// Mitsubishi GX Developer project: パレット取り外し   PLC: Q02

PROGRAM MAIN
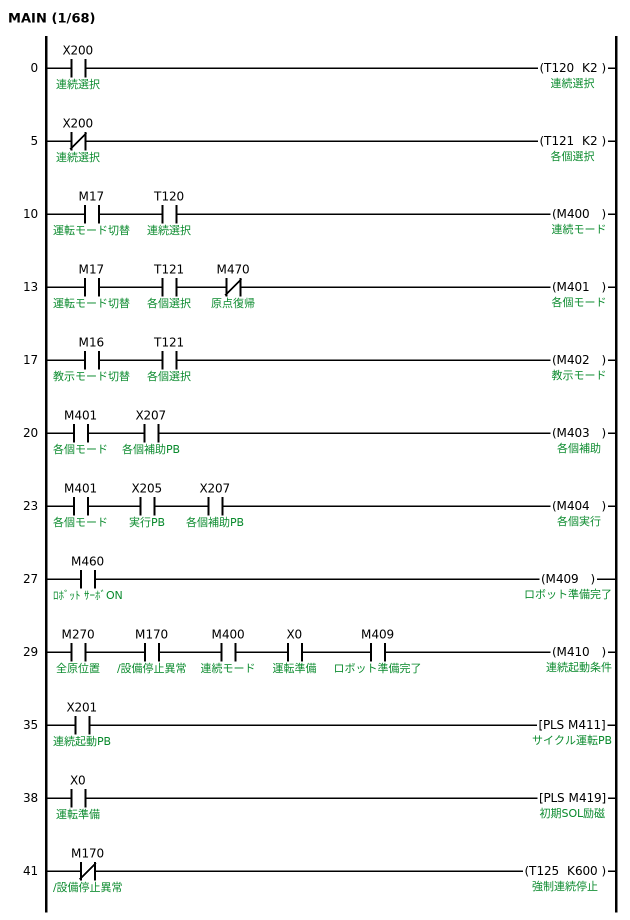
0     LD      X200  ; 連続選択
      OUT     T120 K2  ; 連続選択
5     LDI     X200  ; 連続選択
      OUT     T121 K2  ; 各個選択
10    LD      M17  ; 運転モード切替
      AND     T120  ; 連続選択
      OUT     M400  ; 連続モード
13    LD      M17  ; 運転モード切替
      AND     T121  ; 各個選択
      ANI     M470  ; 原点復帰
      OUT     M401  ; 各個モード
17    LD      M16  ; 教示モード切替
      AND     T121  ; 各個選択
      OUT     M402  ; 教示モード
20    LD      M401  ; 各個モード
      AND     X207  ; 各個補助PB
      OUT     M403  ; 各個補助
23    LD      M401  ; 各個モード
      AND     X205  ; 実行PB
      AND     X207  ; 各個補助PB
      OUT     M404  ; 各個実行
27    LD      M460  ; ﾛﾎﾞｯﾄ ｻｰﾎﾞON
      OUT     M409  ; ロボット準備完了
29    LD      M270  ; 全原位置
      AND     M170  ; /設備停止異常
      AND     M400  ; 連続モード
      AND     X0  ; 運転準備
      AND     M409  ; ロボット準備完了
      OUT     M410  ; 連続起動条件
35    LD      X201  ; 連続起動PB
      PLS     M411  ; サイクル運転PB
38    LD      X0  ; 運転準備
      PLS     M419  ; 初期SOL励磁
41    LDI     M170  ; /設備停止異常
      OUT     T125 K600  ; 強制連続停止
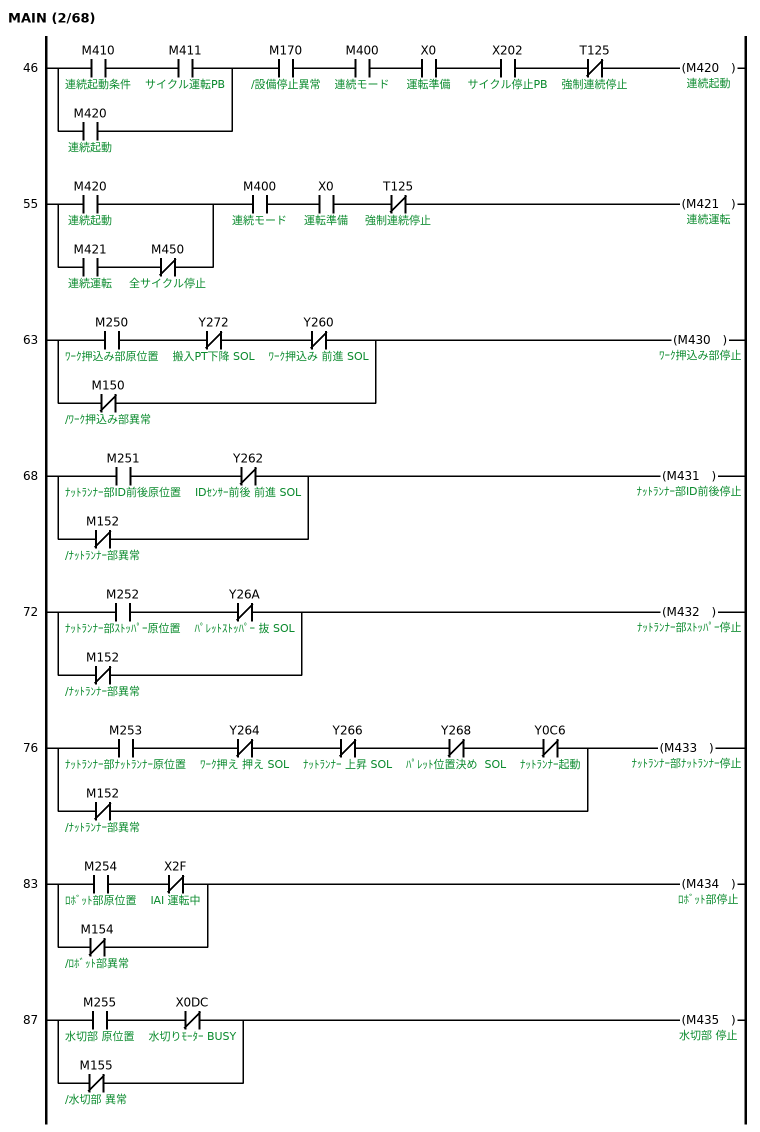
46    LD      M410  ; 連続起動条件
      AND     M411  ; サイクル運転PB
      OR      M420  ; 連続起動
      AND     M170  ; /設備停止異常
      AND     M400  ; 連続モード
      AND     X0  ; 運転準備
      AND     X202  ; サイクル停止PB
      ANI     T125  ; 強制連続停止
      OUT     M420  ; 連続起動
55    LD      M420  ; 連続起動
      LD      M421  ; 連続運転
      ANI     M450  ; 全サイクル停止
      ORB
      AND     M400  ; 連続モード
      AND     X0  ; 運転準備
      ANI     T125  ; 強制連続停止
      OUT     M421  ; 連続運転
63    LD      M250  ; ﾜｰｸ押込み部原位置
      ANI     Y272  ; 搬入PT下降 SOL
      ANI     Y260  ; ﾜｰｸ押込み 前進 SOL
      ORI     M150  ; /ﾜｰｸ押込み部異常
      OUT     M430  ; ﾜｰｸ押込み部停止
68    LD      M251  ; ﾅｯﾄﾗﾝﾅｰ部ID前後原位置
      ANI     Y262  ; IDｾﾝｻｰ前後 前進 SOL
      ORI     M152  ; /ﾅｯﾄﾗﾝﾅｰ部異常
      OUT     M431  ; ﾅｯﾄﾗﾝﾅｰ部ID前後停止
72    LD      M252  ; ﾅｯﾄﾗﾝﾅｰ部ｽﾄｯﾊﾟｰ原位置
      ANI     Y26A  ; ﾊﾟﾚｯﾄｽﾄｯﾊﾟｰ 抜 SOL
      ORI     M152  ; /ﾅｯﾄﾗﾝﾅｰ部異常
      OUT     M432  ; ﾅｯﾄﾗﾝﾅｰ部ｽﾄｯﾊﾟｰ停止
76    LD      M253  ; ﾅｯﾄﾗﾝﾅｰ部ﾅｯﾄﾗﾝﾅｰ原位置
      ANI     Y264  ; ﾜｰｸ押え 押え SOL
      ANI     Y266  ; ﾅｯﾄﾗﾝﾅｰ 上昇 SOL
      ANI     Y268  ; ﾊﾟﾚｯﾄ位置決め  SOL
      ANI     Y0C6  ; ﾅｯﾄﾗﾝﾅｰ起動
      ORI     M152  ; /ﾅｯﾄﾗﾝﾅｰ部異常
      OUT     M433  ; ﾅｯﾄﾗﾝﾅｰ部ﾅｯﾄﾗﾝﾅｰ停止
83    LD      M254  ; ﾛﾎﾞｯﾄ部原位置
      ANI     X2F  ; IAI 運転中
      ORI     M154  ; /ﾛﾎﾞｯﾄ部異常
      OUT     M434  ; ﾛﾎﾞｯﾄ部停止
87    LD      M255  ; 水切部 原位置
      ANI     X0DC  ; 水切りﾓｰﾀｰ BUSY
      ORI     M155  ; /水切部 異常
      OUT     M435  ; 水切部 停止
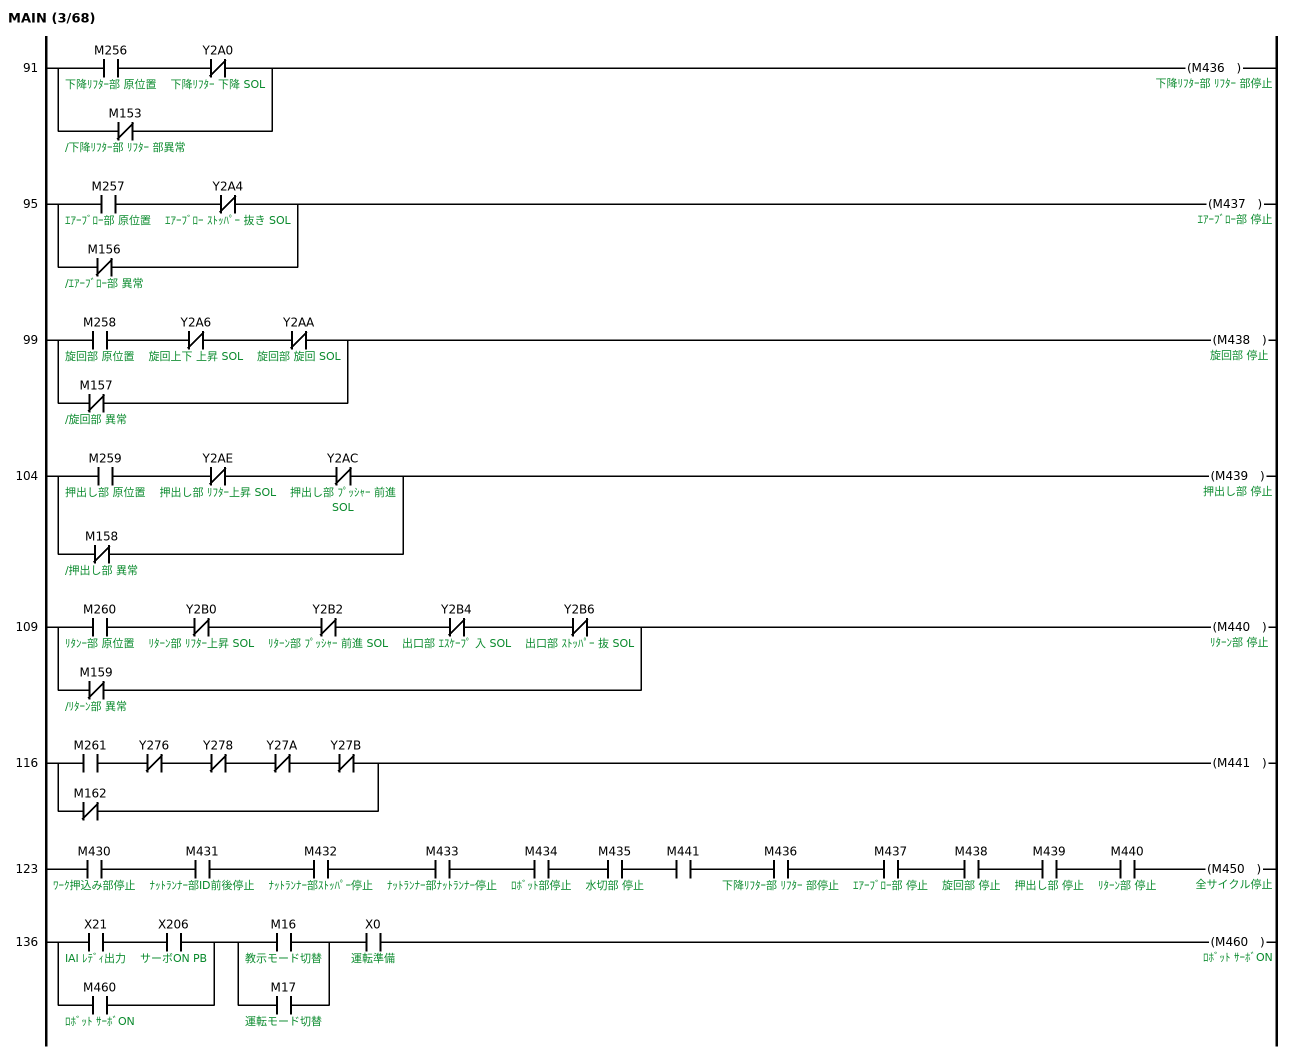
91    LD      M256  ; 下降ﾘﾌﾀｰ部 原位置
      ANI     Y2A0  ; 下降ﾘﾌﾀｰ 下降 SOL
      ORI     M153  ; /下降ﾘﾌﾀｰ部 ﾘﾌﾀｰ 部異常
      OUT     M436  ; 下降ﾘﾌﾀｰ部 ﾘﾌﾀｰ 部停止
95    LD      M257  ; ｴｱｰﾌﾞﾛｰ部 原位置
      ANI     Y2A4  ; ｴｱｰﾌﾞﾛｰ ｽﾄｯﾊﾟｰ 抜き SOL
      ORI     M156  ; /ｴｱｰﾌﾞﾛｰ部 異常
      OUT     M437  ; ｴｱｰﾌﾞﾛｰ部 停止
99    LD      M258  ; 旋回部 原位置
      ANI     Y2A6  ; 旋回上下 上昇 SOL
      ANI     Y2AA  ; 旋回部 旋回 SOL
      ORI     M157  ; /旋回部 異常
      OUT     M438  ; 旋回部 停止
104   LD      M259  ; 押出し部 原位置
      ANI     Y2AE  ; 押出し部 ﾘﾌﾀｰ上昇 SOL
      ANI     Y2AC  ; 押出し部 ﾌﾟｯｼｬｰ 前進 SOL
      ORI     M158  ; /押出し部 異常
      OUT     M439  ; 押出し部 停止
109   LD      M260  ; ﾘﾀﾝｰ部 原位置
      ANI     Y2B0  ; ﾘﾀｰﾝ部 ﾘﾌﾀｰ上昇 SOL
      ANI     Y2B2  ; ﾘﾀｰﾝ部 ﾌﾟｯｼｬｰ 前進 SOL
      ANI     Y2B4  ; 出口部 ｴｽｹｰﾌﾟ 入 SOL
      ANI     Y2B6  ; 出口部 ｽﾄｯﾊﾟｰ 抜 SOL
      ORI     M159  ; /ﾘﾀｰﾝ部 異常
      OUT     M440  ; ﾘﾀｰﾝ部 停止
116   LD      M261
      ANI     Y276
      ANI     Y278
      ANI     Y27A
      ANI     Y27B
      ORI     M162
      OUT     M441
123   LD      M430  ; ﾜｰｸ押込み部停止
      AND     M431  ; ﾅｯﾄﾗﾝﾅｰ部ID前後停止
      AND     M432  ; ﾅｯﾄﾗﾝﾅｰ部ｽﾄｯﾊﾟｰ停止
      AND     M433  ; ﾅｯﾄﾗﾝﾅｰ部ﾅｯﾄﾗﾝﾅｰ停止
      AND     M434  ; ﾛﾎﾞｯﾄ部停止
      AND     M435  ; 水切部 停止
      AND     M441
      AND     M436  ; 下降ﾘﾌﾀｰ部 ﾘﾌﾀｰ 部停止
      AND     M437  ; ｴｱｰﾌﾞﾛｰ部 停止
      AND     M438  ; 旋回部 停止
      AND     M439  ; 押出し部 停止
      AND     M440  ; ﾘﾀｰﾝ部 停止
      OUT     M450  ; 全サイクル停止
136   LD      X21  ; IAI ﾚﾃﾞｨ出力
      AND     X206  ; サーボON PB
      OR      M460  ; ﾛﾎﾞｯﾄ ｻｰﾎﾞON
      LD      M16  ; 教示モード切替
      OR      M17  ; 運転モード切替
      ANB
      AND     X0  ; 運転準備
      OUT     M460  ; ﾛﾎﾞｯﾄ ｻｰﾎﾞON
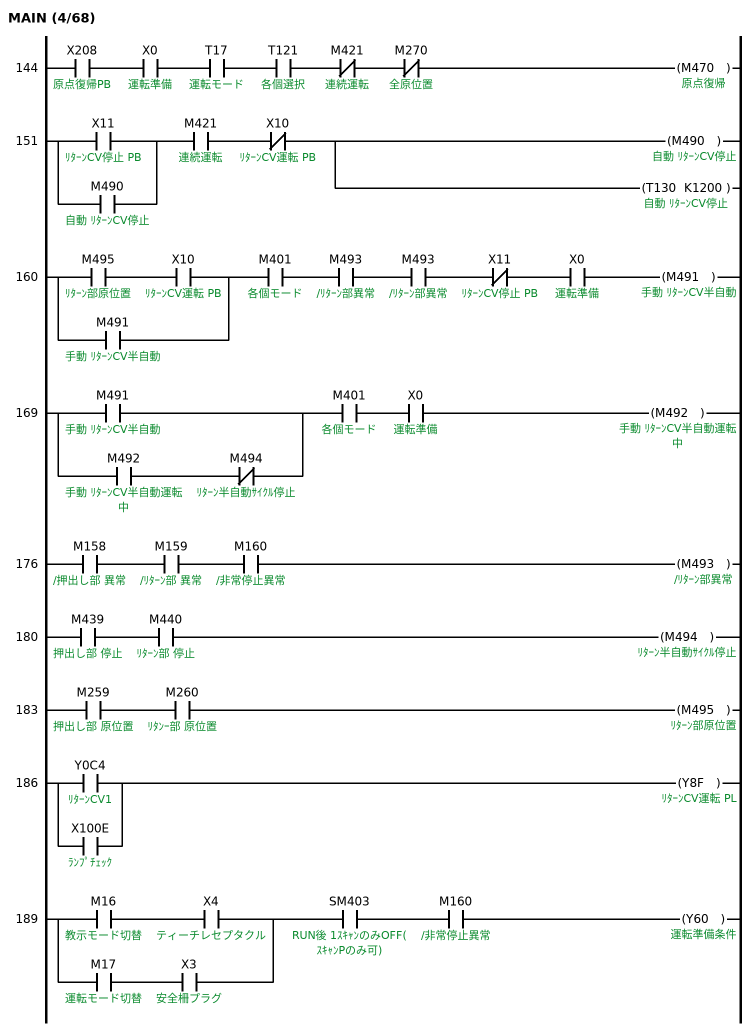
144   LD      X208  ; 原点復帰PB
      AND     X0  ; 運転準備
      AND     T17  ; 運転モード
      AND     T121  ; 各個選択
      ANI     M421  ; 連続運転
      ANI     M270  ; 全原位置
      OUT     M470  ; 原点復帰
151   LD      X11  ; ﾘﾀｰﾝCV停止 PB
      OR      M490  ; 自動 ﾘﾀｰﾝCV停止
      AND     M421  ; 連続運転
      ANI     X10  ; ﾘﾀｰﾝCV運転 PB
      OUT     M490  ; 自動 ﾘﾀｰﾝCV停止
      OUT     T130 K1200  ; 自動 ﾘﾀｰﾝCV停止
160   LD      M495  ; ﾘﾀｰﾝ部原位置
      AND     X10  ; ﾘﾀｰﾝCV運転 PB
      OR      M491  ; 手動 ﾘﾀｰﾝCV半自動
      AND     M401  ; 各個モード
      AND     M493  ; /ﾘﾀｰﾝ部異常
      AND     M493  ; /ﾘﾀｰﾝ部異常
      ANI     X11  ; ﾘﾀｰﾝCV停止 PB
      AND     X0  ; 運転準備
      OUT     M491  ; 手動 ﾘﾀｰﾝCV半自動
169   LD      M491  ; 手動 ﾘﾀｰﾝCV半自動
      LD      M492  ; 手動 ﾘﾀｰﾝCV半自動運転中
      ANI     M494  ; ﾘﾀｰﾝ半自動ｻｲｸﾙ停止
      ORB
      AND     M401  ; 各個モード
      AND     X0  ; 運転準備
      OUT     M492  ; 手動 ﾘﾀｰﾝCV半自動運転中
176   LD      M158  ; /押出し部 異常
      AND     M159  ; /ﾘﾀｰﾝ部 異常
      AND     M160  ; /非常停止異常
      OUT     M493  ; /ﾘﾀｰﾝ部異常
180   LD      M439  ; 押出し部 停止
      AND     M440  ; ﾘﾀｰﾝ部 停止
      OUT     M494  ; ﾘﾀｰﾝ半自動ｻｲｸﾙ停止
183   LD      M259  ; 押出し部 原位置
      AND     M260  ; ﾘﾀﾝｰ部 原位置
      OUT     M495  ; ﾘﾀｰﾝ部原位置
186   LD      Y0C4  ; ﾘﾀｰﾝCV1
      OR      X100E  ; ﾗﾝﾌﾟﾁｪｯｸ
      OUT     Y8F  ; ﾘﾀｰﾝCV運転 PL
189   LD      M16  ; 教示モード切替
      AND     X4  ; ティーチレセプタクル
      LD      M17  ; 運転モード切替
      AND     X3  ; 安全柵プラグ
      ORB
      AND     SM403  ; RUN後 1ｽｷｬﾝのみOFF(ｽｷｬﾝPのみ可)
      AND     M160  ; /非常停止異常
      OUT     Y60  ; 運転準備条件
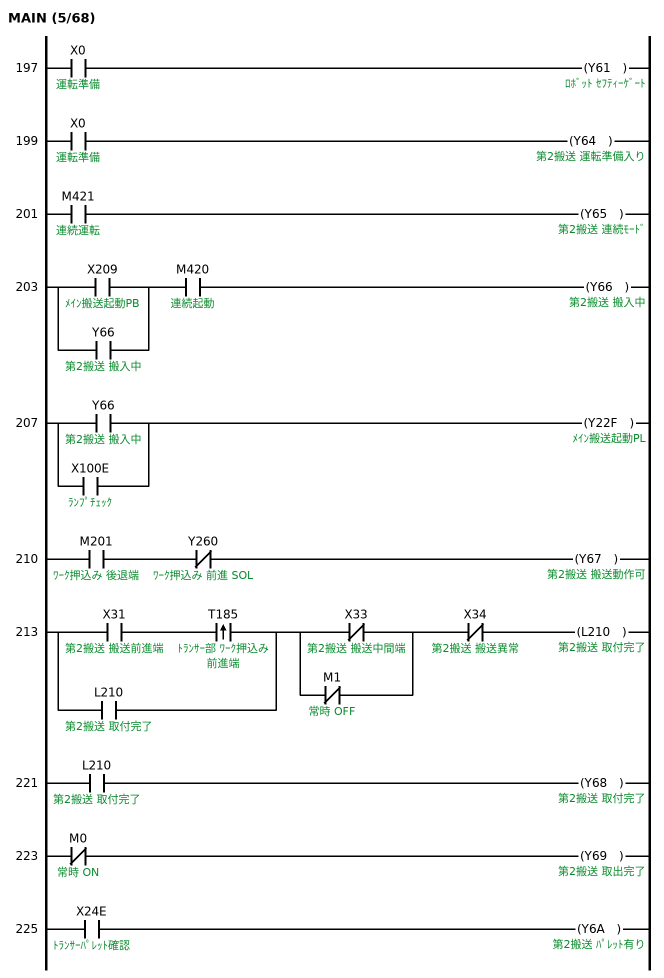
197   LD      X0  ; 運転準備
      OUT     Y61  ; ﾛﾎﾞｯﾄ ｾﾌﾃｨｰｹﾞｰﾄ
199   LD      X0  ; 運転準備
      OUT     Y64  ; 第2搬送 運転準備入り
201   LD      M421  ; 連続運転
      OUT     Y65  ; 第2搬送 連続ﾓｰﾄﾞ
203   LD      X209  ; ﾒｲﾝ搬送起動PB
      OR      Y66  ; 第2搬送 搬入中
      AND     M420  ; 連続起動
      OUT     Y66  ; 第2搬送 搬入中
207   LD      Y66  ; 第2搬送 搬入中
      OR      X100E  ; ﾗﾝﾌﾟﾁｪｯｸ
      OUT     Y22F  ; ﾒｲﾝ搬送起動PL
210   LD      M201  ; ﾜｰｸ押込み 後退端
      ANI     Y260  ; ﾜｰｸ押込み 前進 SOL
      OUT     Y67  ; 第2搬送 搬送動作可
213   LD      X31  ; 第2搬送 搬送前進端
      ANDP    T185  ; ﾄﾗﾝｻｰ部 ﾜｰｸ押込み 前進端
      OR      L210  ; 第2搬送 取付完了
      LDI     X33  ; 第2搬送 搬送中間端
      ORI     M1  ; 常時 OFF
      ANB
      ANI     X34  ; 第2搬送 搬送異常
      OUT     L210  ; 第2搬送 取付完了
221   LD      L210  ; 第2搬送 取付完了
      OUT     Y68  ; 第2搬送 取付完了
223   LDI     M0  ; 常時 ON
      OUT     Y69  ; 第2搬送 取出完了
225   LD      X24E  ; ﾄﾗﾝｻｰﾊﾟﾚｯﾄ確認
      OUT     Y6A  ; 第2搬送 ﾊﾟﾚｯﾄ有り
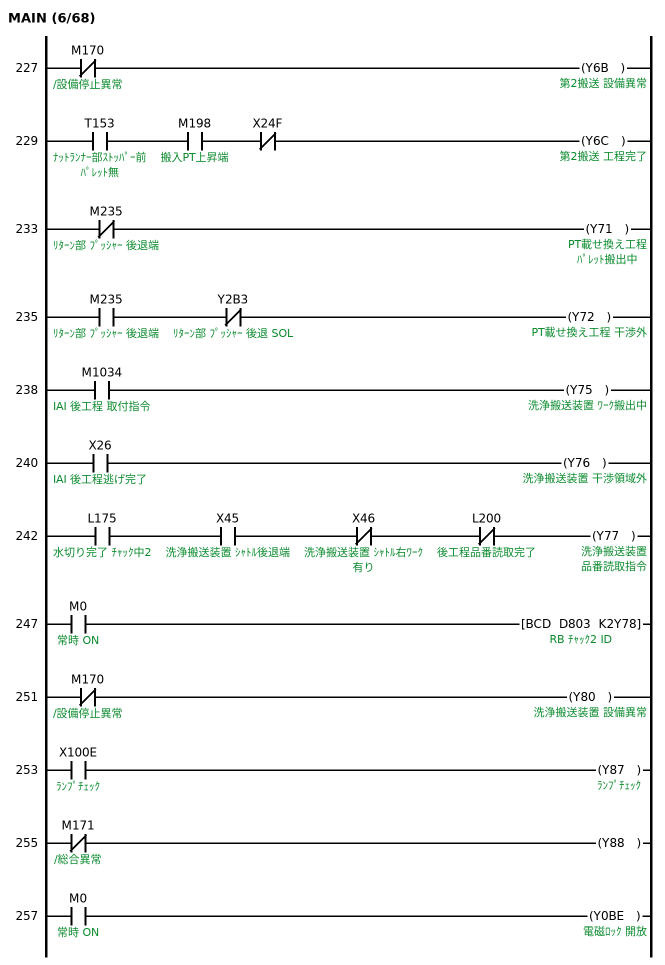
227   LDI     M170  ; /設備停止異常
      OUT     Y6B  ; 第2搬送 設備異常
229   LD      T153  ; ﾅｯﾄﾗﾝﾅｰ部ｽﾄｯﾊﾟｰ前 ﾊﾟﾚｯﾄ無
      AND     M198  ; 搬入PT上昇端
      ANI     X24F
      OUT     Y6C  ; 第2搬送 工程完了
233   LDI     M235  ; ﾘﾀｰﾝ部 ﾌﾟｯｼｬｰ 後退端
      OUT     Y71  ; PT載せ換え工程 ﾊﾟﾚｯﾄ搬出中
235   LD      M235  ; ﾘﾀｰﾝ部 ﾌﾟｯｼｬｰ 後退端
      ANI     Y2B3  ; ﾘﾀｰﾝ部 ﾌﾟｯｼｬｰ 後退 SOL
      OUT     Y72  ; PT載せ換え工程 干渉外
238   LD      M1034  ; IAI 後工程 取付指令
      OUT     Y75  ; 洗浄搬送装置 ﾜｰｸ搬出中
240   LD      X26  ; IAI 後工程逃げ完了
      OUT     Y76  ; 洗浄搬送装置 干渉領域外
242   LD      L175  ; 水切り完了 ﾁｬｯｸ中2
      AND     X45  ; 洗浄搬送装置 ｼｬﾄﾙ後退端
      ANI     X46  ; 洗浄搬送装置 ｼｬﾄﾙ右ﾜｰｸ有り
      ANI     L200  ; 後工程品番読取完了
      OUT     Y77  ; 洗浄搬送装置 品番読取指令
247   LD      M0  ; 常時 ON
      BCD     D803 K2Y78  ; RB ﾁｬｯｸ2 ID / 洗浄搬送装置 品番情報1
251   LDI     M170  ; /設備停止異常
      OUT     Y80  ; 洗浄搬送装置 設備異常
253   LD      X100E  ; ﾗﾝﾌﾟﾁｪｯｸ
      OUT     Y87  ; ﾗﾝﾌﾟﾁｪｯｸ
255   LDI     M171  ; /総合異常
      OUT     Y88
257   LD      M0  ; 常時 ON
      OUT     Y0BE  ; 電磁ﾛｯｸ 開放
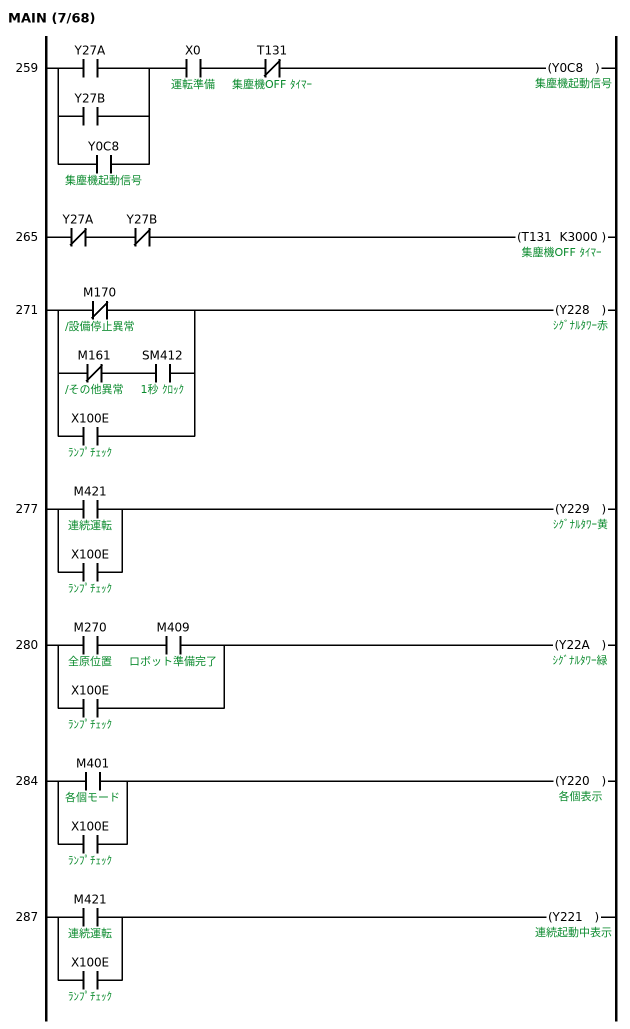
259   LD      Y27A
      OR      Y27B
      OR      Y0C8  ; 集塵機起動信号
      AND     X0  ; 運転準備
      ANI     T131  ; 集塵機OFF ﾀｲﾏｰ
      OUT     Y0C8  ; 集塵機起動信号
265   LDI     Y27A
      ANI     Y27B
      OUT     T131 K3000  ; 集塵機OFF ﾀｲﾏｰ
271   LDI     M170  ; /設備停止異常
      LDI     M161  ; /その他異常
      AND     SM412  ; 1秒 ｸﾛｯｸ
      ORB
      OR      X100E  ; ﾗﾝﾌﾟﾁｪｯｸ
      OUT     Y228  ; ｼｸﾞﾅﾙﾀﾜｰ赤
277   LD      M421  ; 連続運転
      OR      X100E  ; ﾗﾝﾌﾟﾁｪｯｸ
      OUT     Y229  ; ｼｸﾞﾅﾙﾀﾜｰ黄
280   LD      M270  ; 全原位置
      AND     M409  ; ロボット準備完了
      OR      X100E  ; ﾗﾝﾌﾟﾁｪｯｸ
      OUT     Y22A  ; ｼｸﾞﾅﾙﾀﾜｰ緑
284   LD      M401  ; 各個モード
      OR      X100E  ; ﾗﾝﾌﾟﾁｪｯｸ
      OUT     Y220  ; 各個表示
287   LD      M421  ; 連続運転
      OR      X100E  ; ﾗﾝﾌﾟﾁｪｯｸ
      OUT     Y221  ; 連続起動中表示
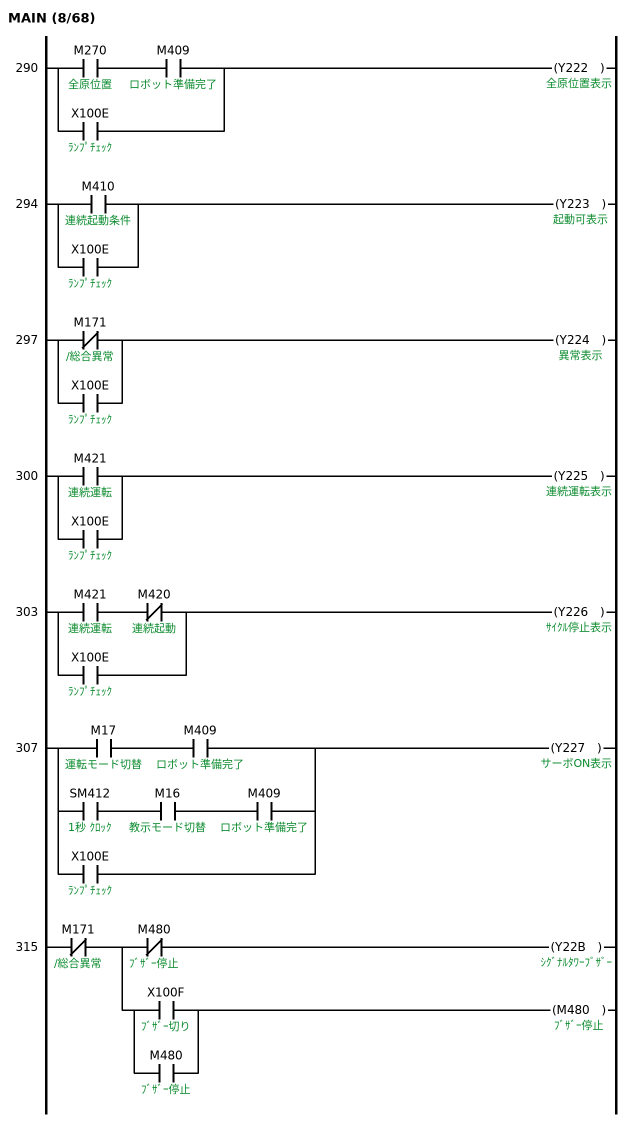
290   LD      M270  ; 全原位置
      AND     M409  ; ロボット準備完了
      OR      X100E  ; ﾗﾝﾌﾟﾁｪｯｸ
      OUT     Y222  ; 全原位置表示
294   LD      M410  ; 連続起動条件
      OR      X100E  ; ﾗﾝﾌﾟﾁｪｯｸ
      OUT     Y223  ; 起動可表示
297   LDI     M171  ; /総合異常
      OR      X100E  ; ﾗﾝﾌﾟﾁｪｯｸ
      OUT     Y224  ; 異常表示
300   LD      M421  ; 連続運転
      OR      X100E  ; ﾗﾝﾌﾟﾁｪｯｸ
      OUT     Y225  ; 連続運転表示
303   LD      M421  ; 連続運転
      ANI     M420  ; 連続起動
      OR      X100E  ; ﾗﾝﾌﾟﾁｪｯｸ
      OUT     Y226  ; ｻｲｸﾙ停止表示
307   LD      M17  ; 運転モード切替
      AND     M409  ; ロボット準備完了
      LD      SM412  ; 1秒 ｸﾛｯｸ
      AND     M16  ; 教示モード切替
      AND     M409  ; ロボット準備完了
      ORB
      OR      X100E  ; ﾗﾝﾌﾟﾁｪｯｸ
      OUT     Y227  ; サーボON表示
315   LDI     M171  ; /総合異常
      MPS
      ANI     M480  ; ﾌﾞｻﾞｰ停止
      OUT     Y22B  ; ｼｸﾞﾅﾙﾀﾜｰﾌﾞｻﾞｰ
      MPP
      LD      X100F  ; ﾌﾞｻﾞｰ切り
      OR      M480  ; ﾌﾞｻﾞｰ停止
      ANB
      OUT     M480  ; ﾌﾞｻﾞｰ停止
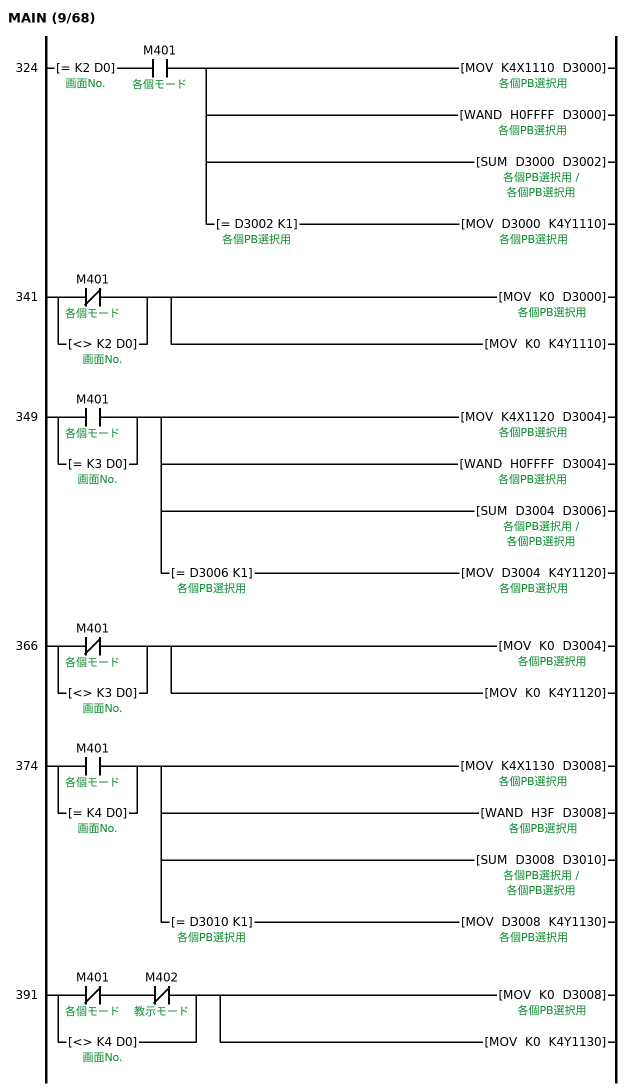
324   LD=     K2 D0  ; 画面No.
      AND     M401  ; 各個モード
      MOV     K4X1110 D3000  ; ﾜｰｸ押込み 後退 PB / 各個PB選択用
      WAND    H0FFFF D3000
      SUM     D3000 D3002  ; 各個PB選択用
      AND=    D3002 K1  ; 各個PB選択用
      MOV     D3000 K4Y1110  ; ﾜｰｸ押込み 後退 選択PL
341   LDI     M401  ; 各個モード
      OR<>    K2 D0  ; 画面No.
      MOV     K0 D3000
      MOV     K0 K4Y1110
349   LD      M401  ; 各個モード
      OR=     K3 D0  ; 画面No.
      MOV     K4X1120 D3004  ; 下降ﾘﾌﾀｰ部 ﾘﾌﾀｰ下降 PB / 各個PB選択用
      WAND    H0FFFF D3004
      SUM     D3004 D3006  ; 各個PB選択用
      AND=    D3006 K1  ; 各個PB選択用
      MOV     D3004 K4Y1120  ; 下降ﾘﾌﾀｰ部 ﾘﾌﾀｰ下降 選択PL
366   LDI     M401  ; 各個モード
      OR<>    K3 D0  ; 画面No.
      MOV     K0 D3004
      MOV     K0 K4Y1120
374   LD      M401  ; 各個モード
      OR=     K4 D0  ; 画面No.
      MOV     K4X1130 D3008  ; ﾛﾎﾞｯﾄ部 ﾁｬｯｸ1開 PB / 各個PB選択用
      WAND    H3F D3008
      SUM     D3008 D3010  ; 各個PB選択用
      AND=    D3010 K1  ; 各個PB選択用
      MOV     D3008 K4Y1130  ; ﾛﾎﾞｯﾄ部 ﾁｬｯｸ1開 選択PL
391   LDI     M401  ; 各個モード
      ANI     M402  ; 教示モード
      OR<>    K4 D0  ; 画面No.
      MOV     K0 D3008
      MOV     K0 K4Y1130
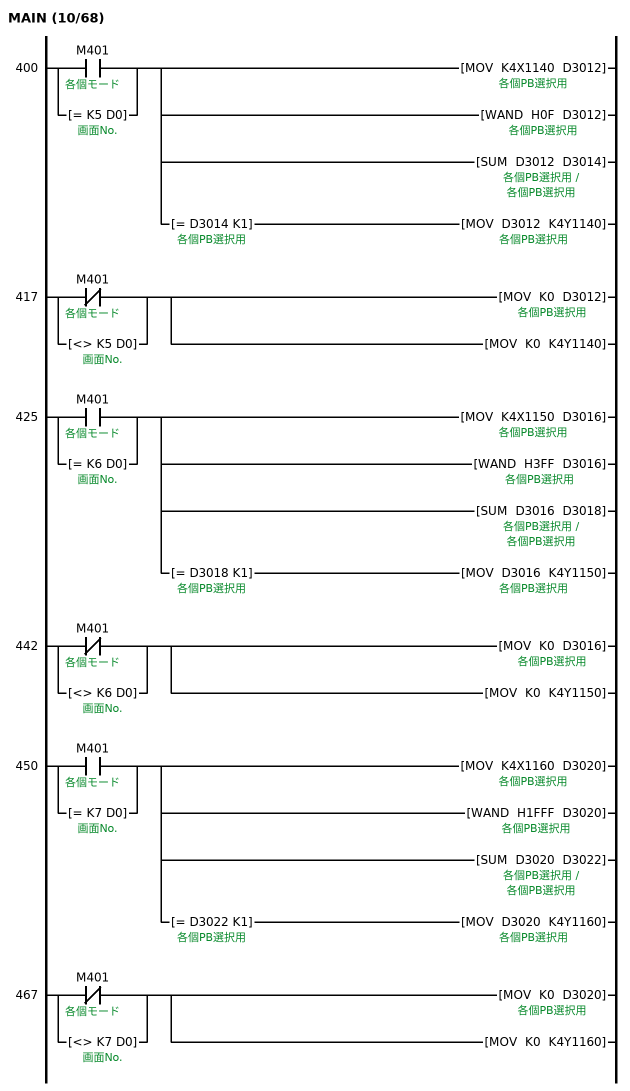
400   LD      M401  ; 各個モード
      OR=     K5 D0  ; 画面No.
      MOV     K4X1140 D3012  ; 水切部 ｼｬｯﾀｰ開 PB / 各個PB選択用
      WAND    H0F D3012
      SUM     D3012 D3014  ; 各個PB選択用
      AND=    D3014 K1  ; 各個PB選択用
      MOV     D3012 K4Y1140  ; 水切部 ｼｬｯﾀｰ開 選択PL
417   LDI     M401  ; 各個モード
      OR<>    K5 D0  ; 画面No.
      MOV     K0 D3012
      MOV     K0 K4Y1140
425   LD      M401  ; 各個モード
      OR=     K6 D0  ; 画面No.
      MOV     K4X1150 D3016  ; ｴｱｰﾌﾞﾛｰ ｼｬｯﾀｰ 開 PB / 各個PB選択用
      WAND    H3FF D3016
      SUM     D3016 D3018  ; 各個PB選択用
      AND=    D3018 K1  ; 各個PB選択用
      MOV     D3016 K4Y1150  ; ｴｱｰﾌﾞﾛｰ ｼｬｯﾀｰ 開 選択PL
442   LDI     M401  ; 各個モード
      OR<>    K6 D0  ; 画面No.
      MOV     K0 D3016
      MOV     K0 K4Y1150
450   LD      M401  ; 各個モード
      OR=     K7 D0  ; 画面No.
      MOV     K4X1160 D3020  ; 押出し部 ﾘﾌﾀｰ下降PB / 各個PB選択用
      WAND    H1FFF D3020
      SUM     D3020 D3022  ; 各個PB選択用
      AND=    D3022 K1  ; 各個PB選択用
      MOV     D3020 K4Y1160  ; 押出し部 ﾘﾌﾀｰ下降選択PL
467   LDI     M401  ; 各個モード
      OR<>    K7 D0  ; 画面No.
      MOV     K0 D3020
      MOV     K0 K4Y1160
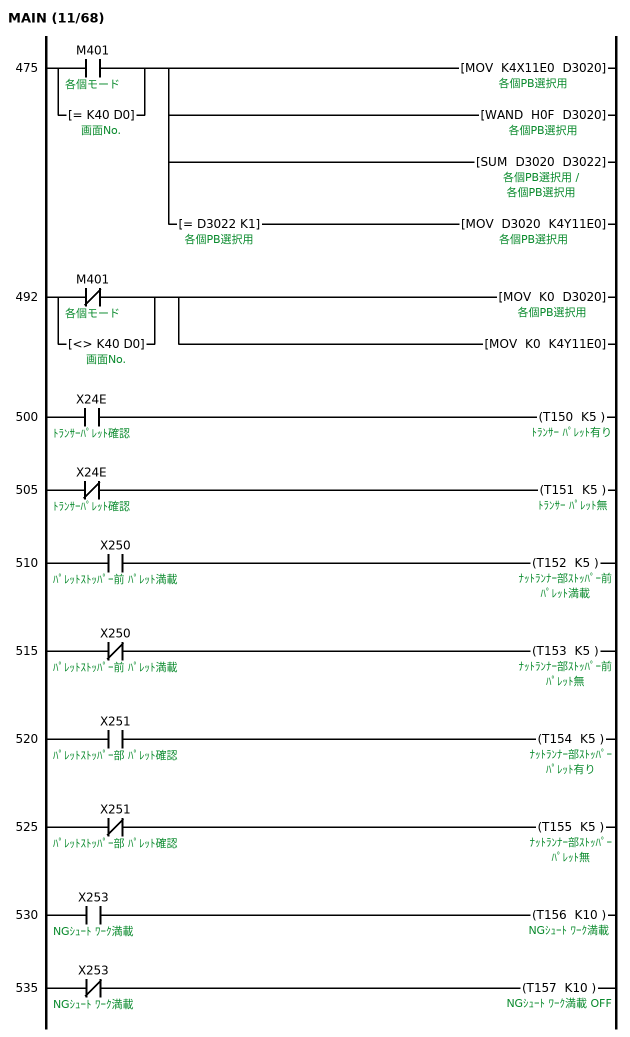
475   LD      M401  ; 各個モード
      OR=     K40 D0  ; 画面No.
      MOV     K4X11E0 D3020  ; ID読出し PB
      WAND    H0F D3020
      SUM     D3020 D3022
      AND=    D3022 K1  ; 各個PB選択用
      MOV     D3020 K4Y11E0  ; ID読出し 選択PL
492   LDI     M401  ; 各個モード
      OR<>    K40 D0  ; 画面No.
      MOV     K0 D3020
      MOV     K0 K4Y11E0
500   LD      X24E  ; ﾄﾗﾝｻｰﾊﾟﾚｯﾄ確認
      OUT     T150 K5  ; ﾄﾗﾝｻｰ ﾊﾟﾚｯﾄ有り
505   LDI     X24E  ; ﾄﾗﾝｻｰﾊﾟﾚｯﾄ確認
      OUT     T151 K5  ; ﾄﾗﾝｻｰ ﾊﾟﾚｯﾄ無
510   LD      X250  ; ﾊﾟﾚｯﾄｽﾄｯﾊﾟｰ前 ﾊﾟﾚｯﾄ満載
      OUT     T152 K5  ; ﾅｯﾄﾗﾝﾅｰ部ｽﾄｯﾊﾟｰ前 ﾊﾟﾚｯﾄ満載
515   LDI     X250  ; ﾊﾟﾚｯﾄｽﾄｯﾊﾟｰ前 ﾊﾟﾚｯﾄ満載
      OUT     T153 K5  ; ﾅｯﾄﾗﾝﾅｰ部ｽﾄｯﾊﾟｰ前 ﾊﾟﾚｯﾄ無
520   LD      X251  ; ﾊﾟﾚｯﾄｽﾄｯﾊﾟｰ部 ﾊﾟﾚｯﾄ確認
      OUT     T154 K5  ; ﾅｯﾄﾗﾝﾅｰ部ｽﾄｯﾊﾟｰ ﾊﾟﾚｯﾄ有り
525   LDI     X251  ; ﾊﾟﾚｯﾄｽﾄｯﾊﾟｰ部 ﾊﾟﾚｯﾄ確認
      OUT     T155 K5  ; ﾅｯﾄﾗﾝﾅｰ部ｽﾄｯﾊﾟｰ ﾊﾟﾚｯﾄ無
530   LD      X253  ; NGｼｭｰﾄ ﾜｰｸ満載
      OUT     T156 K10  ; NGｼｭｰﾄ ﾜｰｸ満載
535   LDI     X253  ; NGｼｭｰﾄ ﾜｰｸ満載
      OUT     T157 K10  ; NGｼｭｰﾄ ﾜｰｸ満載 OFF
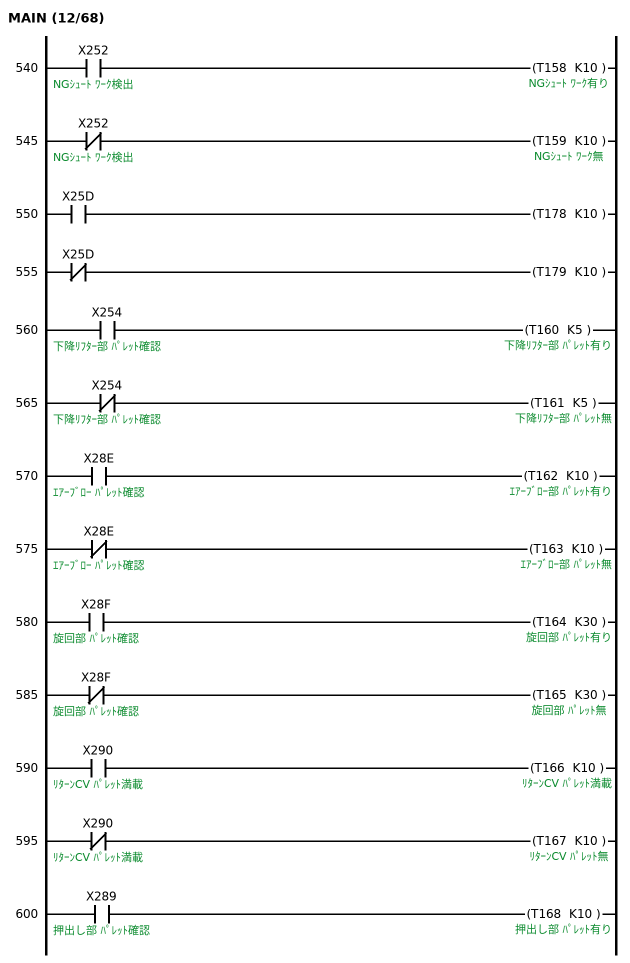
540   LD      X252  ; NGｼｭｰﾄ ﾜｰｸ検出
      OUT     T158 K10  ; NGｼｭｰﾄ ﾜｰｸ有り
545   LDI     X252  ; NGｼｭｰﾄ ﾜｰｸ検出
      OUT     T159 K10  ; NGｼｭｰﾄ ﾜｰｸ無
550   LD      X25D
      OUT     T178 K10
555   LDI     X25D
      OUT     T179 K10
560   LD      X254  ; 下降ﾘﾌﾀｰ部 ﾊﾟﾚｯﾄ確認
      OUT     T160 K5  ; 下降ﾘﾌﾀｰ部 ﾊﾟﾚｯﾄ有り
565   LDI     X254  ; 下降ﾘﾌﾀｰ部 ﾊﾟﾚｯﾄ確認
      OUT     T161 K5  ; 下降ﾘﾌﾀｰ部 ﾊﾟﾚｯﾄ無
570   LD      X28E  ; ｴｱｰﾌﾞﾛｰ ﾊﾟﾚｯﾄ確認
      OUT     T162 K10  ; ｴｱｰﾌﾞﾛｰ部 ﾊﾟﾚｯﾄ有り
575   LDI     X28E  ; ｴｱｰﾌﾞﾛｰ ﾊﾟﾚｯﾄ確認
      OUT     T163 K10  ; ｴｱｰﾌﾞﾛｰ部 ﾊﾟﾚｯﾄ無
580   LD      X28F  ; 旋回部 ﾊﾟﾚｯﾄ確認
      OUT     T164 K30  ; 旋回部 ﾊﾟﾚｯﾄ有り
585   LDI     X28F  ; 旋回部 ﾊﾟﾚｯﾄ確認
      OUT     T165 K30  ; 旋回部 ﾊﾟﾚｯﾄ無
590   LD      X290  ; ﾘﾀｰﾝCV ﾊﾟﾚｯﾄ満載
      OUT     T166 K10  ; ﾘﾀｰﾝCV ﾊﾟﾚｯﾄ満載
595   LDI     X290  ; ﾘﾀｰﾝCV ﾊﾟﾚｯﾄ満載
      OUT     T167 K10  ; ﾘﾀｰﾝCV ﾊﾟﾚｯﾄ無
600   LD      X289  ; 押出し部 ﾊﾟﾚｯﾄ確認
      OUT     T168 K10  ; 押出し部 ﾊﾟﾚｯﾄ有り
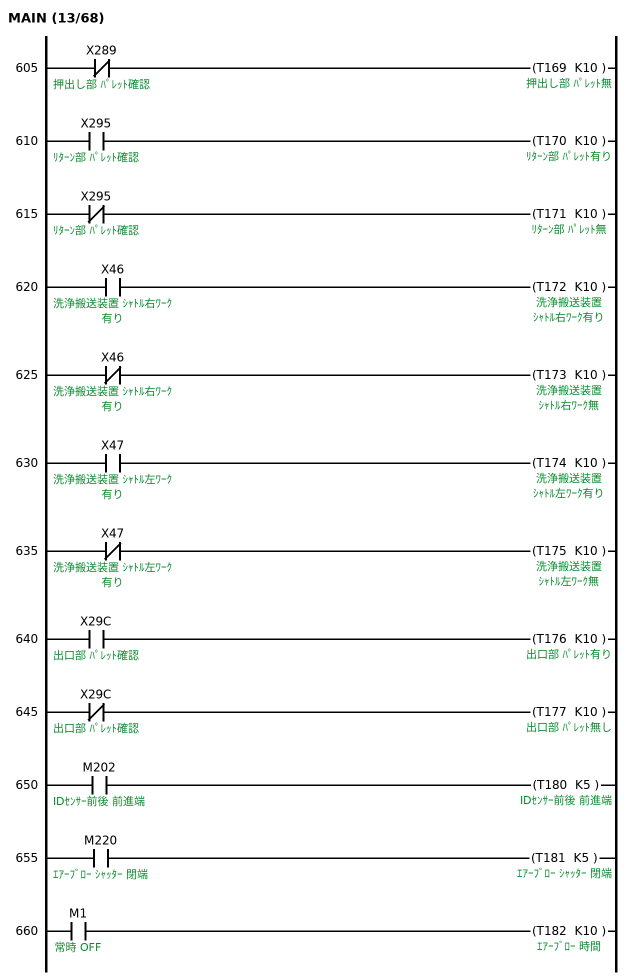
605   LDI     X289  ; 押出し部 ﾊﾟﾚｯﾄ確認
      OUT     T169 K10  ; 押出し部 ﾊﾟﾚｯﾄ無
610   LD      X295  ; ﾘﾀｰﾝ部 ﾊﾟﾚｯﾄ確認
      OUT     T170 K10  ; ﾘﾀｰﾝ部 ﾊﾟﾚｯﾄ有り
615   LDI     X295  ; ﾘﾀｰﾝ部 ﾊﾟﾚｯﾄ確認
      OUT     T171 K10  ; ﾘﾀｰﾝ部 ﾊﾟﾚｯﾄ無
620   LD      X46  ; 洗浄搬送装置 ｼｬﾄﾙ右ﾜｰｸ有り
      OUT     T172 K10  ; 洗浄搬送装置 ｼｬﾄﾙ右ﾜｰｸ有り
625   LDI     X46  ; 洗浄搬送装置 ｼｬﾄﾙ右ﾜｰｸ有り
      OUT     T173 K10  ; 洗浄搬送装置 ｼｬﾄﾙ右ﾜｰｸ無
630   LD      X47  ; 洗浄搬送装置 ｼｬﾄﾙ左ﾜｰｸ有り
      OUT     T174 K10  ; 洗浄搬送装置 ｼｬﾄﾙ左ﾜｰｸ有り
635   LDI     X47  ; 洗浄搬送装置 ｼｬﾄﾙ左ﾜｰｸ有り
      OUT     T175 K10  ; 洗浄搬送装置 ｼｬﾄﾙ左ﾜｰｸ無
640   LD      X29C  ; 出口部 ﾊﾟﾚｯﾄ確認
      OUT     T176 K10  ; 出口部 ﾊﾟﾚｯﾄ有り
645   LDI     X29C  ; 出口部 ﾊﾟﾚｯﾄ確認
      OUT     T177 K10  ; 出口部 ﾊﾟﾚｯﾄ無し
650   LD      M202  ; IDｾﾝｻｰ前後 前進端
      OUT     T180 K5  ; IDｾﾝｻｰ前後 前進端
655   LD      M220  ; ｴｱｰﾌﾞﾛｰ ｼｬｯﾀｰ 閉端
      OUT     T181 K5  ; ｴｱｰﾌﾞﾛｰ ｼｬｯﾀｰ 閉端
660   LD      M1  ; 常時 OFF
      OUT     T182 K10  ; ｴｱｰﾌﾞﾛｰ 時間
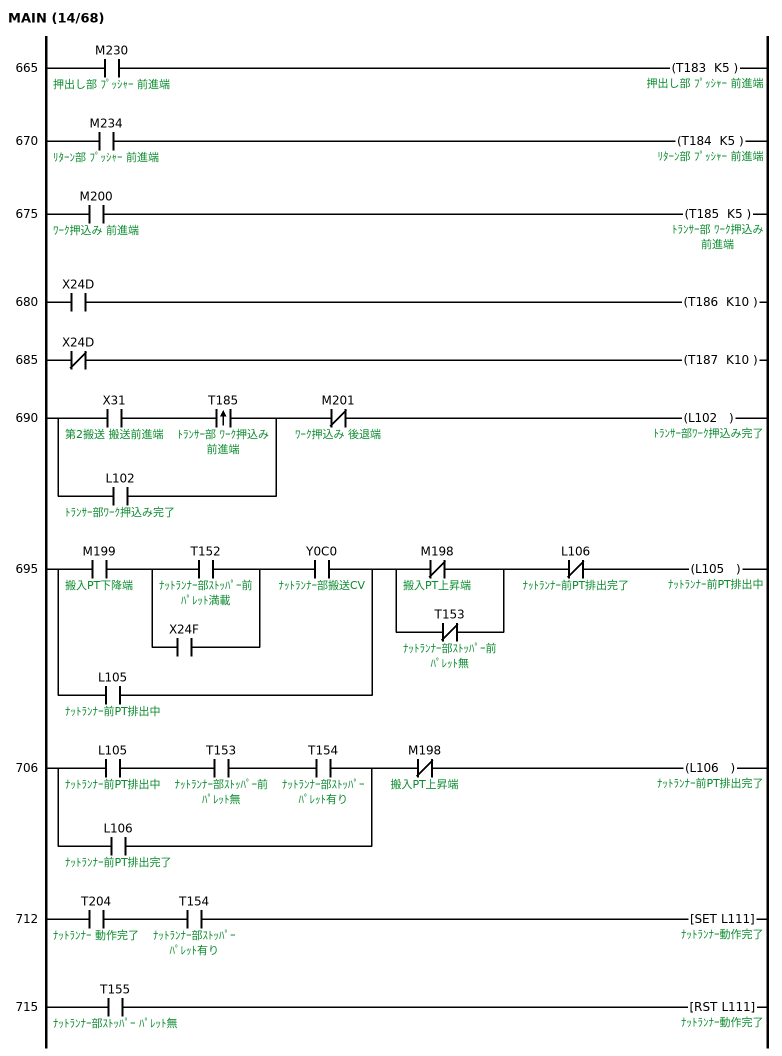
665   LD      M230  ; 押出し部 ﾌﾟｯｼｬｰ 前進端
      OUT     T183 K5  ; 押出し部 ﾌﾟｯｼｬｰ 前進端
670   LD      M234  ; ﾘﾀｰﾝ部 ﾌﾟｯｼｬｰ 前進端
      OUT     T184 K5  ; ﾘﾀｰﾝ部 ﾌﾟｯｼｬｰ 前進端
675   LD      M200  ; ﾜｰｸ押込み 前進端
      OUT     T185 K5  ; ﾄﾗﾝｻｰ部 ﾜｰｸ押込み 前進端
680   LD      X24D
      OUT     T186 K10
685   LDI     X24D
      OUT     T187 K10
690   LD      X31  ; 第2搬送 搬送前進端
      ANDP    T185  ; ﾄﾗﾝｻｰ部 ﾜｰｸ押込み 前進端
      OR      L102  ; ﾄﾗﾝｻｰ部ﾜｰｸ押込み完了
      ANI     M201  ; ﾜｰｸ押込み 後退端
      OUT     L102  ; ﾄﾗﾝｻｰ部ﾜｰｸ押込み完了
695   LD      M199  ; 搬入PT下降端
      LD      T152  ; ﾅｯﾄﾗﾝﾅｰ部ｽﾄｯﾊﾟｰ前 ﾊﾟﾚｯﾄ満載
      OR      X24F
      ANB
      AND     Y0C0  ; ﾅｯﾄﾗﾝﾅｰ部搬送CV
      OR      L105  ; ﾅｯﾄﾗﾝﾅｰ前PT排出中
      LDI     M198  ; 搬入PT上昇端
      ORI     T153  ; ﾅｯﾄﾗﾝﾅｰ部ｽﾄｯﾊﾟｰ前 ﾊﾟﾚｯﾄ無
      ANB
      ANI     L106  ; ﾅｯﾄﾗﾝﾅｰ前PT排出完了
      OUT     L105  ; ﾅｯﾄﾗﾝﾅｰ前PT排出中
706   LD      L105  ; ﾅｯﾄﾗﾝﾅｰ前PT排出中
      AND     T153  ; ﾅｯﾄﾗﾝﾅｰ部ｽﾄｯﾊﾟｰ前 ﾊﾟﾚｯﾄ無
      AND     T154  ; ﾅｯﾄﾗﾝﾅｰ部ｽﾄｯﾊﾟｰ ﾊﾟﾚｯﾄ有り
      OR      L106  ; ﾅｯﾄﾗﾝﾅｰ前PT排出完了
      ANI     M198  ; 搬入PT上昇端
      OUT     L106  ; ﾅｯﾄﾗﾝﾅｰ前PT排出完了
712   LD      T204  ; ﾅｯﾄﾗﾝﾅｰ 動作完了
      AND     T154  ; ﾅｯﾄﾗﾝﾅｰ部ｽﾄｯﾊﾟｰ ﾊﾟﾚｯﾄ有り
      SET     L111  ; ﾅｯﾄﾗﾝﾅｰ動作完了
715   LD      T155  ; ﾅｯﾄﾗﾝﾅｰ部ｽﾄｯﾊﾟｰ ﾊﾟﾚｯﾄ無
      RST     L111  ; ﾅｯﾄﾗﾝﾅｰ動作完了
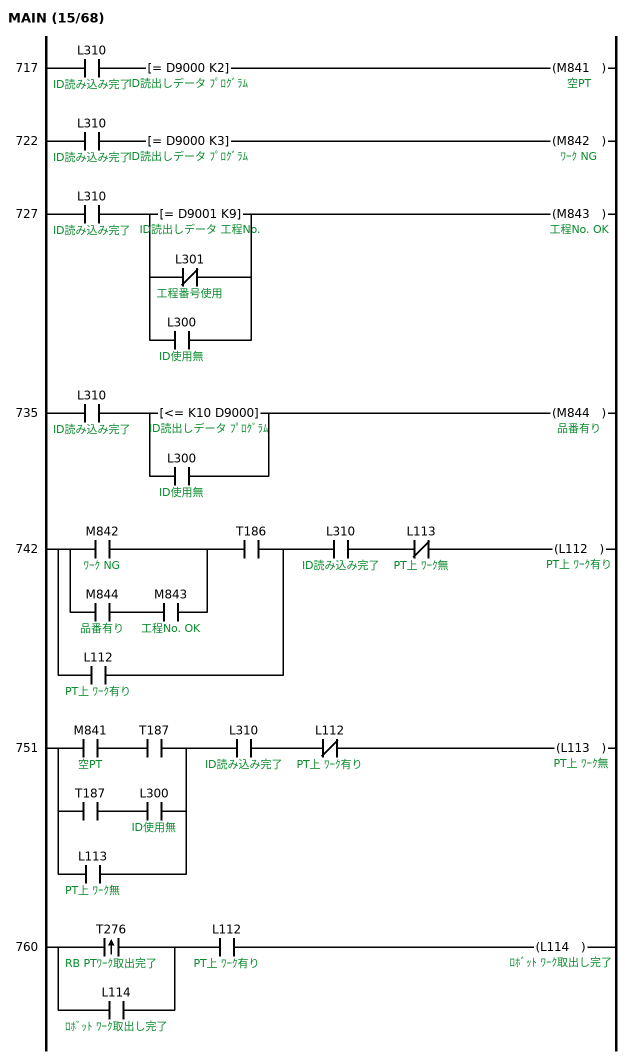
717   LD      L310  ; ID読み込み完了
      AND=    D9000 K2  ; ID読出しデータ ﾌﾟﾛｸﾞﾗﾑ
      OUT     M841  ; 空PT
722   LD      L310  ; ID読み込み完了
      AND=    D9000 K3  ; ID読出しデータ ﾌﾟﾛｸﾞﾗﾑ
      OUT     M842  ; ﾜｰｸ NG
727   LD      L310  ; ID読み込み完了
      LD=     D9001 K9  ; ID読出しデータ 工程No.
      ORI     L301  ; 工程番号使用
      OR      L300  ; ID使用無
      ANB
      OUT     M843  ; 工程No. OK
735   LD      L310  ; ID読み込み完了
      LD<=    K10 D9000  ; ID読出しデータ ﾌﾟﾛｸﾞﾗﾑ
      OR      L300  ; ID使用無
      ANB
      OUT     M844  ; 品番有り
742   LD      M842  ; ﾜｰｸ NG
      LD      M844  ; 品番有り
      AND     M843  ; 工程No. OK
      ORB
      AND     T186
      OR      L112  ; PT上 ﾜｰｸ有り
      AND     L310  ; ID読み込み完了
      ANI     L113  ; PT上 ﾜｰｸ無
      OUT     L112  ; PT上 ﾜｰｸ有り
751   LD      M841  ; 空PT
      AND     T187
      LD      T187
      AND     L300  ; ID使用無
      ORB
      OR      L113  ; PT上 ﾜｰｸ無
      AND     L310  ; ID読み込み完了
      ANI     L112  ; PT上 ﾜｰｸ有り
      OUT     L113  ; PT上 ﾜｰｸ無
760   LDP     T276  ; RB PTﾜｰｸ取出完了
      OR      L114  ; ﾛﾎﾞｯﾄ ﾜｰｸ取出し完了
      AND     L112  ; PT上 ﾜｰｸ有り
      OUT     L114  ; ﾛﾎﾞｯﾄ ﾜｰｸ取出し完了
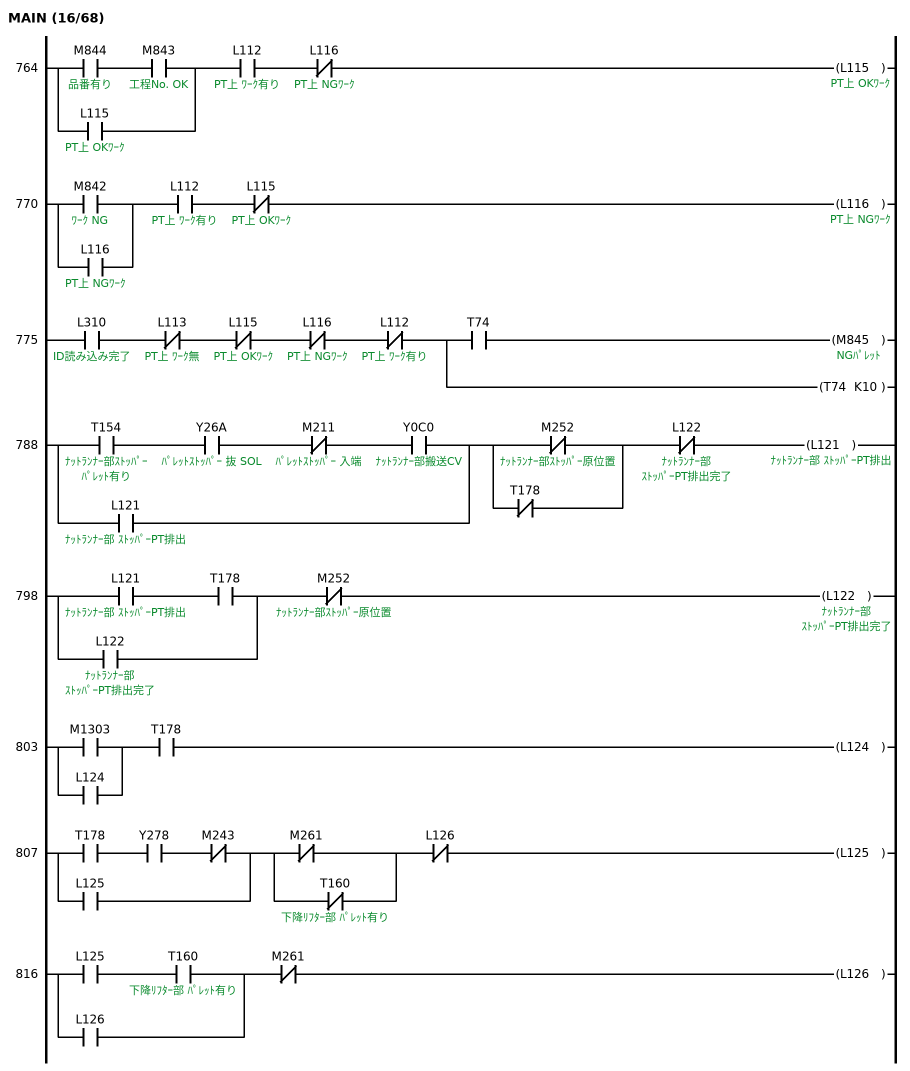
764   LD      M844  ; 品番有り
      AND     M843  ; 工程No. OK
      OR      L115  ; PT上 OKﾜｰｸ
      AND     L112  ; PT上 ﾜｰｸ有り
      ANI     L116  ; PT上 NGﾜｰｸ
      OUT     L115  ; PT上 OKﾜｰｸ
770   LD      M842  ; ﾜｰｸ NG
      OR      L116  ; PT上 NGﾜｰｸ
      AND     L112  ; PT上 ﾜｰｸ有り
      ANI     L115  ; PT上 OKﾜｰｸ
      OUT     L116  ; PT上 NGﾜｰｸ
775   LD      L310  ; ID読み込み完了
      ANI     L113  ; PT上 ﾜｰｸ無
      ANI     L115  ; PT上 OKﾜｰｸ
      ANI     L116  ; PT上 NGﾜｰｸ
      ANI     L112  ; PT上 ﾜｰｸ有り
      MPS
      AND     T74
      OUT     M845  ; NGﾊﾟﾚｯﾄ
      MPP
      OUT     T74 K10
788   LD      T154  ; ﾅｯﾄﾗﾝﾅｰ部ｽﾄｯﾊﾟｰ ﾊﾟﾚｯﾄ有り
      AND     Y26A  ; ﾊﾟﾚｯﾄｽﾄｯﾊﾟｰ 抜 SOL
      ANI     M211  ; ﾊﾟﾚｯﾄｽﾄｯﾊﾟｰ 入端
      AND     Y0C0  ; ﾅｯﾄﾗﾝﾅｰ部搬送CV
      OR      L121  ; ﾅｯﾄﾗﾝﾅｰ部 ｽﾄｯﾊﾟｰPT排出
      LDI     M252  ; ﾅｯﾄﾗﾝﾅｰ部ｽﾄｯﾊﾟｰ原位置
      ORI     T178
      ANB
      ANI     L122  ; ﾅｯﾄﾗﾝﾅｰ部 ｽﾄｯﾊﾟｰPT排出完了
      OUT     L121  ; ﾅｯﾄﾗﾝﾅｰ部 ｽﾄｯﾊﾟｰPT排出
798   LD      L121  ; ﾅｯﾄﾗﾝﾅｰ部 ｽﾄｯﾊﾟｰPT排出
      AND     T178
      OR      L122  ; ﾅｯﾄﾗﾝﾅｰ部 ｽﾄｯﾊﾟｰPT排出完了
      ANI     M252  ; ﾅｯﾄﾗﾝﾅｰ部ｽﾄｯﾊﾟｰ原位置
      OUT     L122  ; ﾅｯﾄﾗﾝﾅｰ部 ｽﾄｯﾊﾟｰPT排出完了
803   LD      M1303
      OR      L124
      AND     T178
      OUT     L124
807   LD      T178
      AND     Y278
      ANI     M243
      OR      L125
      LDI     M261
      ORI     T160  ; 下降ﾘﾌﾀｰ部 ﾊﾟﾚｯﾄ有り
      ANB
      ANI     L126
      OUT     L125
816   LD      L125
      AND     T160  ; 下降ﾘﾌﾀｰ部 ﾊﾟﾚｯﾄ有り
      OR      L126
      ANI     M261
      OUT     L126
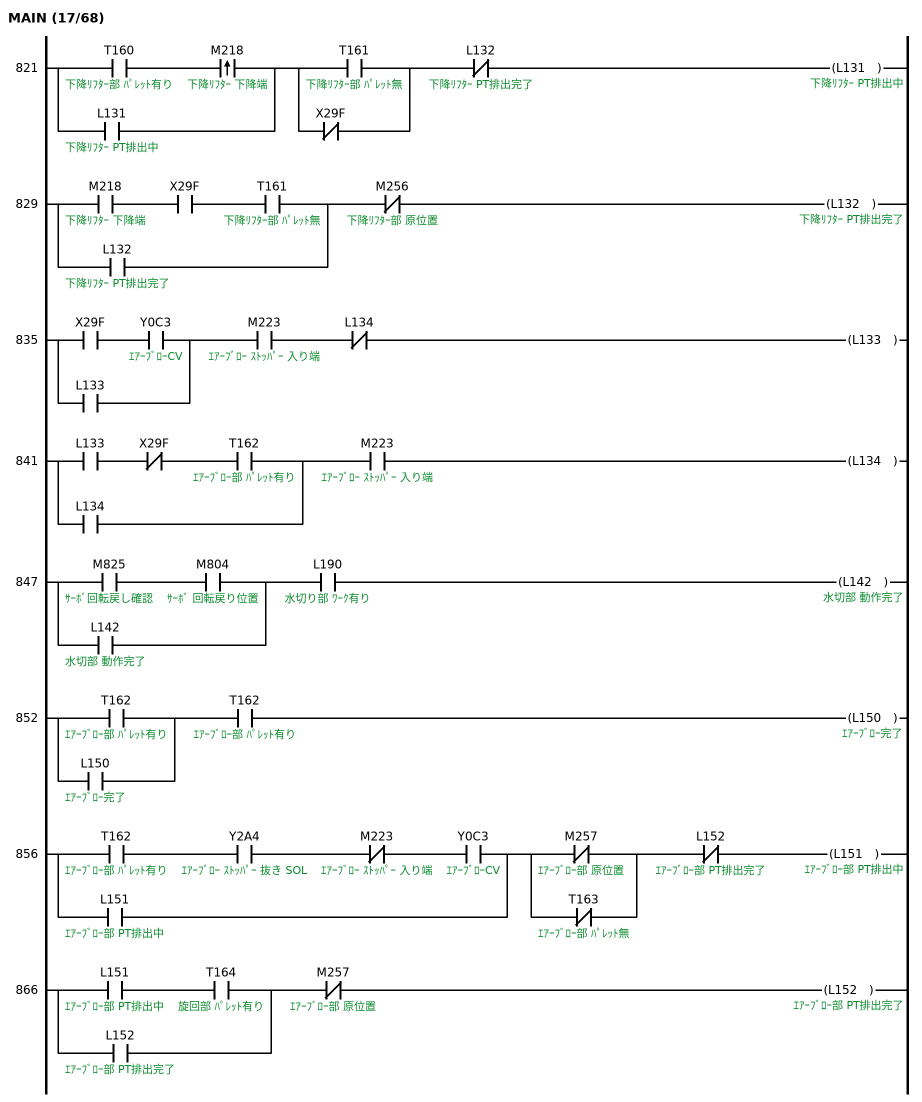
821   LD      T160  ; 下降ﾘﾌﾀｰ部 ﾊﾟﾚｯﾄ有り
      ANDP    M218  ; 下降ﾘﾌﾀｰ 下降端
      OR      L131  ; 下降ﾘﾌﾀｰ PT排出中
      LD      T161  ; 下降ﾘﾌﾀｰ部 ﾊﾟﾚｯﾄ無
      ORI     X29F
      ANB
      ANI     L132  ; 下降ﾘﾌﾀｰ PT排出完了
      OUT     L131  ; 下降ﾘﾌﾀｰ PT排出中
829   LD      M218  ; 下降ﾘﾌﾀｰ 下降端
      AND     X29F
      AND     T161  ; 下降ﾘﾌﾀｰ部 ﾊﾟﾚｯﾄ無
      OR      L132  ; 下降ﾘﾌﾀｰ PT排出完了
      ANI     M256  ; 下降ﾘﾌﾀｰ部 原位置
      OUT     L132  ; 下降ﾘﾌﾀｰ PT排出完了
835   LD      X29F
      AND     Y0C3  ; ｴｱｰﾌﾞﾛｰCV
      OR      L133
      AND     M223  ; ｴｱｰﾌﾞﾛｰ ｽﾄｯﾊﾟｰ 入り端
      ANI     L134
      OUT     L133
841   LD      L133
      ANI     X29F
      AND     T162  ; ｴｱｰﾌﾞﾛｰ部 ﾊﾟﾚｯﾄ有り
      OR      L134
      AND     M223  ; ｴｱｰﾌﾞﾛｰ ｽﾄｯﾊﾟｰ 入り端
      OUT     L134
847   LD      M825  ; ｻｰﾎﾞ回転戻し確認
      AND     M804  ; ｻｰﾎﾞ 回転戻り位置
      OR      L142  ; 水切部 動作完了
      AND     L190  ; 水切り部 ﾜｰｸ有り
      OUT     L142  ; 水切部 動作完了
852   LD      T162  ; ｴｱｰﾌﾞﾛｰ部 ﾊﾟﾚｯﾄ有り
      OR      L150  ; ｴｱｰﾌﾞﾛｰ完了
      AND     T162  ; ｴｱｰﾌﾞﾛｰ部 ﾊﾟﾚｯﾄ有り
      OUT     L150  ; ｴｱｰﾌﾞﾛｰ完了
856   LD      T162  ; ｴｱｰﾌﾞﾛｰ部 ﾊﾟﾚｯﾄ有り
      AND     Y2A4  ; ｴｱｰﾌﾞﾛｰ ｽﾄｯﾊﾟｰ 抜き SOL
      ANI     M223  ; ｴｱｰﾌﾞﾛｰ ｽﾄｯﾊﾟｰ 入り端
      AND     Y0C3  ; ｴｱｰﾌﾞﾛｰCV
      OR      L151  ; ｴｱｰﾌﾞﾛｰ部 PT排出中
      LDI     M257  ; ｴｱｰﾌﾞﾛｰ部 原位置
      ORI     T163  ; ｴｱｰﾌﾞﾛｰ部 ﾊﾟﾚｯﾄ無
      ANB
      ANI     L152  ; ｴｱｰﾌﾞﾛｰ部 PT排出完了
      OUT     L151  ; ｴｱｰﾌﾞﾛｰ部 PT排出中
866   LD      L151  ; ｴｱｰﾌﾞﾛｰ部 PT排出中
      AND     T164  ; 旋回部 ﾊﾟﾚｯﾄ有り
      OR      L152  ; ｴｱｰﾌﾞﾛｰ部 PT排出完了
      ANI     M257  ; ｴｱｰﾌﾞﾛｰ部 原位置
      OUT     L152  ; ｴｱｰﾌﾞﾛｰ部 PT排出完了
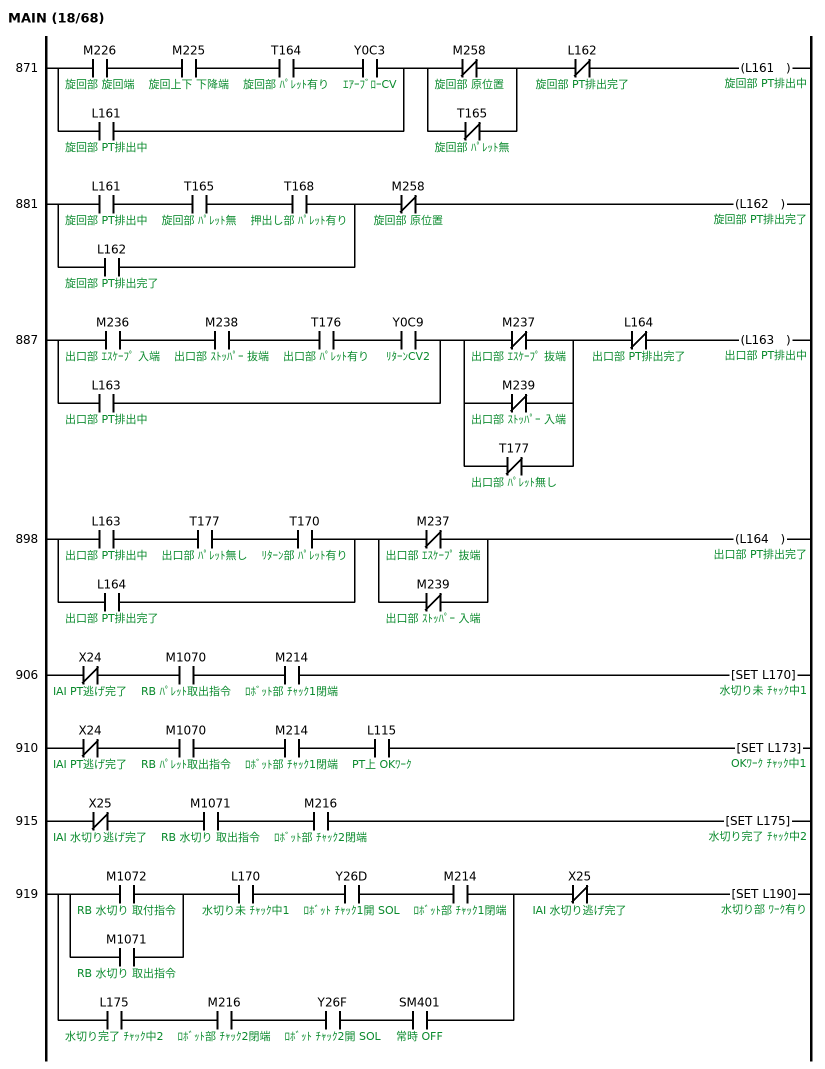
871   LD      M226  ; 旋回部 旋回端
      AND     M225  ; 旋回上下 下降端
      AND     T164  ; 旋回部 ﾊﾟﾚｯﾄ有り
      AND     Y0C3  ; ｴｱｰﾌﾞﾛｰCV
      OR      L161  ; 旋回部 PT排出中
      LDI     M258  ; 旋回部 原位置
      ORI     T165  ; 旋回部 ﾊﾟﾚｯﾄ無
      ANB
      ANI     L162  ; 旋回部 PT排出完了
      OUT     L161  ; 旋回部 PT排出中
881   LD      L161  ; 旋回部 PT排出中
      AND     T165  ; 旋回部 ﾊﾟﾚｯﾄ無
      AND     T168  ; 押出し部 ﾊﾟﾚｯﾄ有り
      OR      L162  ; 旋回部 PT排出完了
      ANI     M258  ; 旋回部 原位置
      OUT     L162  ; 旋回部 PT排出完了
887   LD      M236  ; 出口部 ｴｽｹｰﾌﾟ 入端
      AND     M238  ; 出口部 ｽﾄｯﾊﾟｰ 抜端
      AND     T176  ; 出口部 ﾊﾟﾚｯﾄ有り
      AND     Y0C9  ; ﾘﾀｰﾝCV2
      OR      L163  ; 出口部 PT排出中
      LDI     M237  ; 出口部 ｴｽｹｰﾌﾟ 抜端
      ORI     M239  ; 出口部 ｽﾄｯﾊﾟｰ 入端
      ORI     T177  ; 出口部 ﾊﾟﾚｯﾄ無し
      ANB
      ANI     L164  ; 出口部 PT排出完了
      OUT     L163  ; 出口部 PT排出中
898   LD      L163  ; 出口部 PT排出中
      AND     T177  ; 出口部 ﾊﾟﾚｯﾄ無し
      AND     T170  ; ﾘﾀｰﾝ部 ﾊﾟﾚｯﾄ有り
      OR      L164  ; 出口部 PT排出完了
      LDI     M237  ; 出口部 ｴｽｹｰﾌﾟ 抜端
      ORI     M239  ; 出口部 ｽﾄｯﾊﾟｰ 入端
      ANB
      OUT     L164  ; 出口部 PT排出完了
906   LDI     X24  ; IAI PT逃げ完了
      AND     M1070  ; RB ﾊﾟﾚｯﾄ取出指令
      AND     M214  ; ﾛﾎﾞｯﾄ部 ﾁｬｯｸ1閉端
      SET     L170  ; 水切り未 ﾁｬｯｸ中1
910   LDI     X24  ; IAI PT逃げ完了
      AND     M1070  ; RB ﾊﾟﾚｯﾄ取出指令
      AND     M214  ; ﾛﾎﾞｯﾄ部 ﾁｬｯｸ1閉端
      AND     L115  ; PT上 OKﾜｰｸ
      SET     L173  ; OKﾜｰｸ ﾁｬｯｸ中1
915   LDI     X25  ; IAI 水切り逃げ完了
      AND     M1071  ; RB 水切り 取出指令
      AND     M216  ; ﾛﾎﾞｯﾄ部 ﾁｬｯｸ2閉端
      SET     L175  ; 水切り完了 ﾁｬｯｸ中2
919   LD      M1072  ; RB 水切り 取付指令
      OR      M1071  ; RB 水切り 取出指令
      AND     L170  ; 水切り未 ﾁｬｯｸ中1
      AND     Y26D  ; ﾛﾎﾞｯﾄ ﾁｬｯｸ1開 SOL
      AND     M214  ; ﾛﾎﾞｯﾄ部 ﾁｬｯｸ1閉端
      LD      L175  ; 水切り完了 ﾁｬｯｸ中2
      AND     M216  ; ﾛﾎﾞｯﾄ部 ﾁｬｯｸ2閉端
      AND     Y26F  ; ﾛﾎﾞｯﾄ ﾁｬｯｸ2開 SOL
      AND     SM401  ; 常時 OFF
      ORB
      ANI     X25  ; IAI 水切り逃げ完了
      SET     L190  ; 水切り部 ﾜｰｸ有り
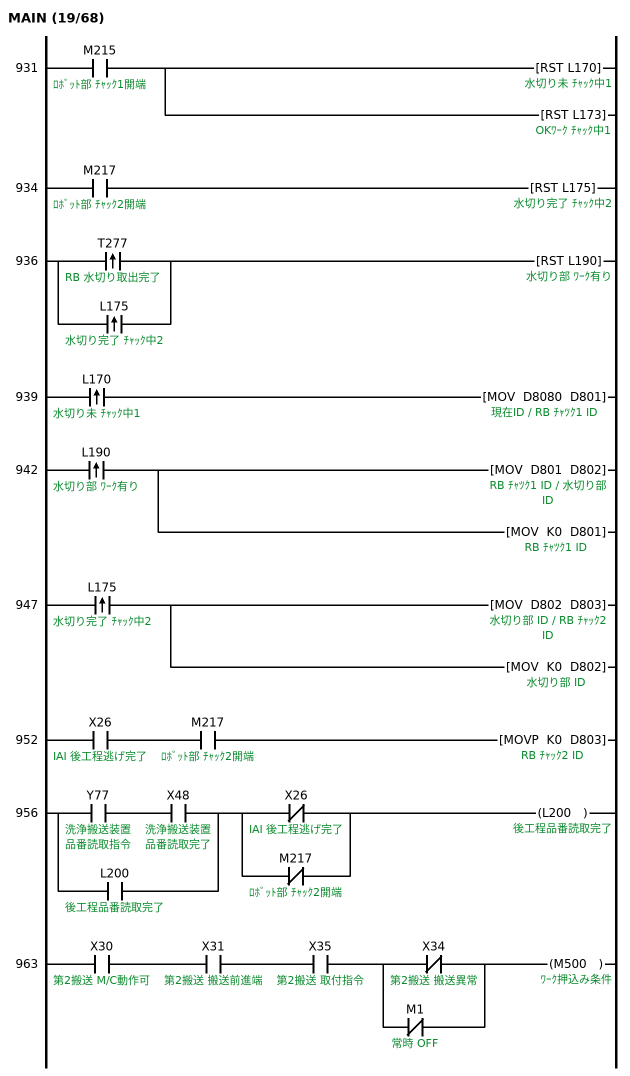
931   LD      M215  ; ﾛﾎﾞｯﾄ部 ﾁｬｯｸ1開端
      RST     L170  ; 水切り未 ﾁｬｯｸ中1
      RST     L173  ; OKﾜｰｸ ﾁｬｯｸ中1
934   LD      M217  ; ﾛﾎﾞｯﾄ部 ﾁｬｯｸ2開端
      RST     L175  ; 水切り完了 ﾁｬｯｸ中2
936   LDP     T277  ; RB 水切り取出完了
      ORP     L175  ; 水切り完了 ﾁｬｯｸ中2
      RST     L190  ; 水切り部 ﾜｰｸ有り
939   LDP     L170  ; 水切り未 ﾁｬｯｸ中1
      MOV     D8080 D801  ; 現在ID / RB ﾁｬﾂｸ1 ID
942   LDP     L190  ; 水切り部 ﾜｰｸ有り
      MOV     D801 D802  ; 水切り部 ID
      MOV     K0 D801
947   LDP     L175  ; 水切り完了 ﾁｬｯｸ中2
      MOV     D802 D803
      MOV     K0 D802
952   LD      X26  ; IAI 後工程逃げ完了
      AND     M217  ; ﾛﾎﾞｯﾄ部 ﾁｬｯｸ2開端
      MOVP    K0 D803
956   LD      Y77  ; 洗浄搬送装置 品番読取指令
      AND     X48  ; 洗浄搬送装置 品番読取完了
      OR      L200  ; 後工程品番読取完了
      LDI     X26  ; IAI 後工程逃げ完了
      ORI     M217  ; ﾛﾎﾞｯﾄ部 ﾁｬｯｸ2開端
      ANB
      OUT     L200  ; 後工程品番読取完了
963   LD      X30  ; 第2搬送 M/C動作可
      AND     X31  ; 第2搬送 搬送前進端
      AND     X35  ; 第2搬送 取付指令
      LDI     X34  ; 第2搬送 搬送異常
      ORI     M1  ; 常時 OFF
      ANB
      OUT     M500  ; ﾜｰｸ押込み条件
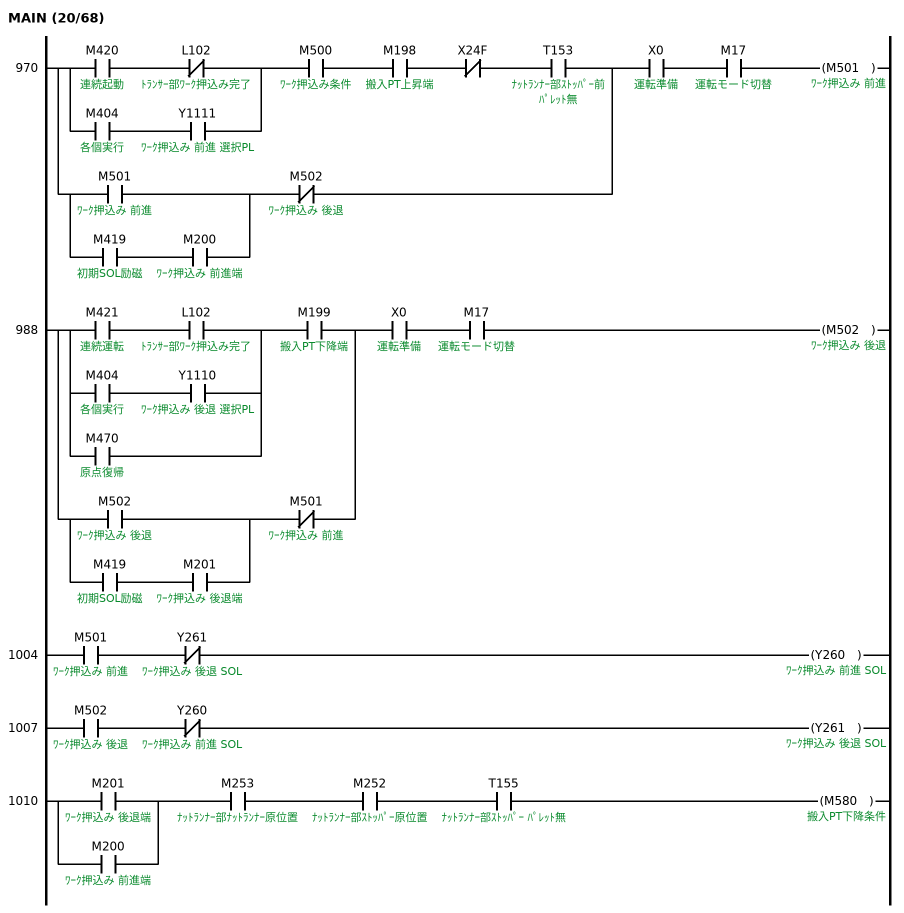
970   LD      M420  ; 連続起動
      ANI     L102  ; ﾄﾗﾝｻｰ部ﾜｰｸ押込み完了
      LD      M404  ; 各個実行
      AND     Y1111  ; ﾜｰｸ押込み 前進 選択PL
      ORB
      AND     M500  ; ﾜｰｸ押込み条件
      AND     M198  ; 搬入PT上昇端
      ANI     X24F
      AND     T153  ; ﾅｯﾄﾗﾝﾅｰ部ｽﾄｯﾊﾟｰ前 ﾊﾟﾚｯﾄ無
      LD      M501  ; ﾜｰｸ押込み 前進
      LD      M419  ; 初期SOL励磁
      AND     M200  ; ﾜｰｸ押込み 前進端
      ORB
      ANI     M502  ; ﾜｰｸ押込み 後退
      ORB
      AND     X0  ; 運転準備
      AND     M17  ; 運転モード切替
      OUT     M501  ; ﾜｰｸ押込み 前進
988   LD      M421  ; 連続運転
      AND     L102  ; ﾄﾗﾝｻｰ部ﾜｰｸ押込み完了
      LD      M404  ; 各個実行
      AND     Y1110  ; ﾜｰｸ押込み 後退 選択PL
      ORB
      OR      M470  ; 原点復帰
      AND     M199  ; 搬入PT下降端
      LD      M502  ; ﾜｰｸ押込み 後退
      LD      M419  ; 初期SOL励磁
      AND     M201  ; ﾜｰｸ押込み 後退端
      ORB
      ANI     M501  ; ﾜｰｸ押込み 前進
      ORB
      AND     X0  ; 運転準備
      AND     M17  ; 運転モード切替
      OUT     M502  ; ﾜｰｸ押込み 後退
1004  LD      M501  ; ﾜｰｸ押込み 前進
      ANI     Y261  ; ﾜｰｸ押込み 後退 SOL
      OUT     Y260  ; ﾜｰｸ押込み 前進 SOL
1007  LD      M502  ; ﾜｰｸ押込み 後退
      ANI     Y260  ; ﾜｰｸ押込み 前進 SOL
      OUT     Y261  ; ﾜｰｸ押込み 後退 SOL
1010  LD      M201  ; ﾜｰｸ押込み 後退端
      OR      M200  ; ﾜｰｸ押込み 前進端
      AND     M253  ; ﾅｯﾄﾗﾝﾅｰ部ﾅｯﾄﾗﾝﾅｰ原位置
      AND     M252  ; ﾅｯﾄﾗﾝﾅｰ部ｽﾄｯﾊﾟｰ原位置
      AND     T155  ; ﾅｯﾄﾗﾝﾅｰ部ｽﾄｯﾊﾟｰ ﾊﾟﾚｯﾄ無
      OUT     M580  ; 搬入PT下降条件
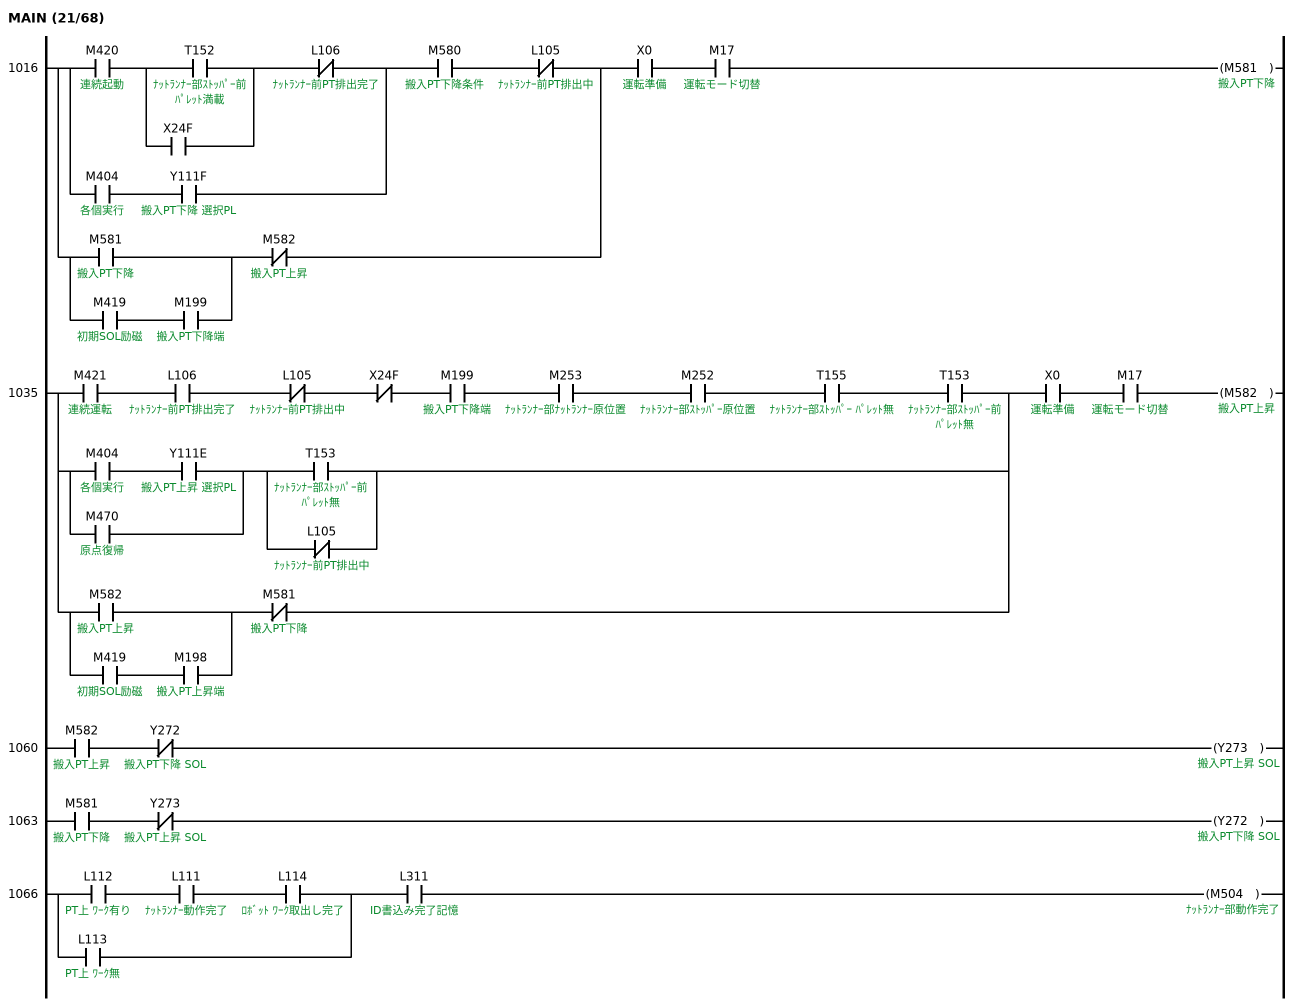
1016  LD      M420  ; 連続起動
      LD      T152  ; ﾅｯﾄﾗﾝﾅｰ部ｽﾄｯﾊﾟｰ前 ﾊﾟﾚｯﾄ満載
      OR      X24F
      ANB
      ANI     L106  ; ﾅｯﾄﾗﾝﾅｰ前PT排出完了
      LD      M404  ; 各個実行
      AND     Y111F  ; 搬入PT下降 選択PL
      ORB
      AND     M580  ; 搬入PT下降条件
      ANI     L105  ; ﾅｯﾄﾗﾝﾅｰ前PT排出中
      LD      M581  ; 搬入PT下降
      LD      M419  ; 初期SOL励磁
      AND     M199  ; 搬入PT下降端
      ORB
      ANI     M582  ; 搬入PT上昇
      ORB
      AND     X0  ; 運転準備
      AND     M17  ; 運転モード切替
      OUT     M581  ; 搬入PT下降
1035  LD      M421  ; 連続運転
      AND     L106  ; ﾅｯﾄﾗﾝﾅｰ前PT排出完了
      ANI     L105  ; ﾅｯﾄﾗﾝﾅｰ前PT排出中
      ANI     X24F
      AND     M199  ; 搬入PT下降端
      AND     M253  ; ﾅｯﾄﾗﾝﾅｰ部ﾅｯﾄﾗﾝﾅｰ原位置
      AND     M252  ; ﾅｯﾄﾗﾝﾅｰ部ｽﾄｯﾊﾟｰ原位置
      AND     T155  ; ﾅｯﾄﾗﾝﾅｰ部ｽﾄｯﾊﾟｰ ﾊﾟﾚｯﾄ無
      AND     T153  ; ﾅｯﾄﾗﾝﾅｰ部ｽﾄｯﾊﾟｰ前 ﾊﾟﾚｯﾄ無
      LD      M404  ; 各個実行
      AND     Y111E  ; 搬入PT上昇 選択PL
      OR      M470  ; 原点復帰
      LD      T153  ; ﾅｯﾄﾗﾝﾅｰ部ｽﾄｯﾊﾟｰ前 ﾊﾟﾚｯﾄ無
      ORI     L105  ; ﾅｯﾄﾗﾝﾅｰ前PT排出中
      ANB
      ORB
      LD      M582  ; 搬入PT上昇
      LD      M419  ; 初期SOL励磁
      AND     M198  ; 搬入PT上昇端
      ORB
      ANI     M581  ; 搬入PT下降
      ORB
      AND     X0  ; 運転準備
      AND     M17  ; 運転モード切替
      OUT     M582  ; 搬入PT上昇
1060  LD      M582  ; 搬入PT上昇
      ANI     Y272  ; 搬入PT下降 SOL
      OUT     Y273  ; 搬入PT上昇 SOL
1063  LD      M581  ; 搬入PT下降
      ANI     Y273  ; 搬入PT上昇 SOL
      OUT     Y272  ; 搬入PT下降 SOL
1066  LD      L112  ; PT上 ﾜｰｸ有り
      AND     L111  ; ﾅｯﾄﾗﾝﾅｰ動作完了
      AND     L114  ; ﾛﾎﾞｯﾄ ﾜｰｸ取出し完了
      OR      L113  ; PT上 ﾜｰｸ無
      AND     L311  ; ID書込み完了記憶
      OUT     M504  ; ﾅｯﾄﾗﾝﾅｰ部動作完了
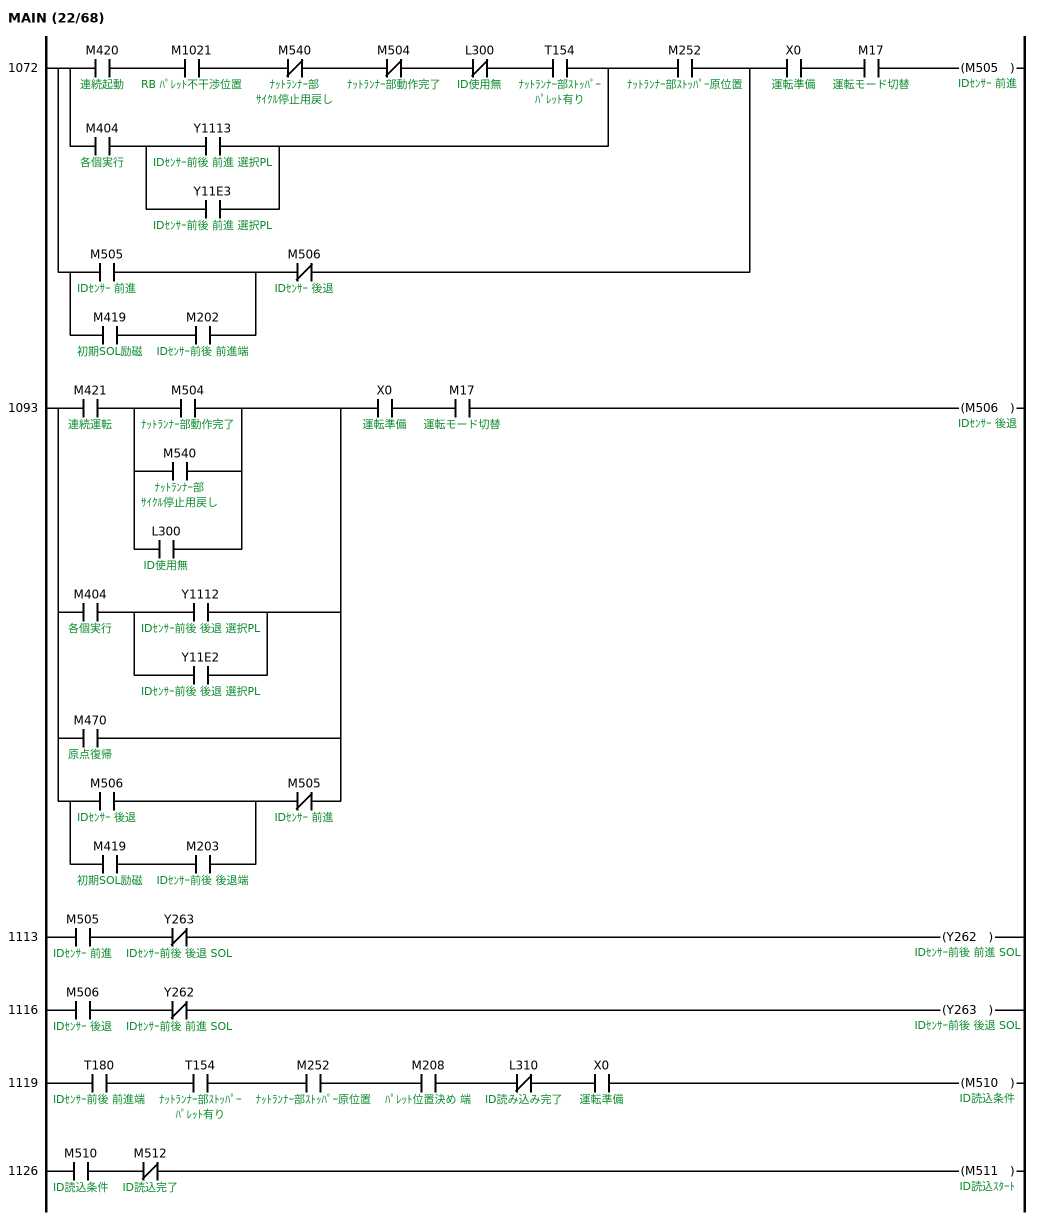
1072  LD      M420  ; 連続起動
      AND     M1021  ; RB ﾊﾟﾚｯﾄ不干渉位置
      ANI     M540  ; ﾅｯﾄﾗﾝﾅｰ部 ｻｲｸﾙ停止用戻し
      ANI     M504  ; ﾅｯﾄﾗﾝﾅｰ部動作完了
      ANI     L300  ; ID使用無
      AND     T154  ; ﾅｯﾄﾗﾝﾅｰ部ｽﾄｯﾊﾟｰ ﾊﾟﾚｯﾄ有り
      LD      M404  ; 各個実行
      LD      Y1113  ; IDｾﾝｻｰ前後 前進 選択PL
      OR      Y11E3  ; IDｾﾝｻｰ前後 前進 選択PL
      ANB
      ORB
      AND     M252  ; ﾅｯﾄﾗﾝﾅｰ部ｽﾄｯﾊﾟｰ原位置
      LD      M505  ; IDｾﾝｻｰ 前進
      LD      M419  ; 初期SOL励磁
      AND     M202  ; IDｾﾝｻｰ前後 前進端
      ORB
      ANI     M506  ; IDｾﾝｻｰ 後退
      ORB
      AND     X0  ; 運転準備
      AND     M17  ; 運転モード切替
      OUT     M505  ; IDｾﾝｻｰ 前進
1093  LD      M421  ; 連続運転
      LD      M504  ; ﾅｯﾄﾗﾝﾅｰ部動作完了
      OR      M540  ; ﾅｯﾄﾗﾝﾅｰ部 ｻｲｸﾙ停止用戻し
      OR      L300  ; ID使用無
      ANB
      LD      M404  ; 各個実行
      LD      Y1112  ; IDｾﾝｻｰ前後 後退 選択PL
      OR      Y11E2  ; IDｾﾝｻｰ前後 後退 選択PL
      ANB
      ORB
      OR      M470  ; 原点復帰
      LD      M506  ; IDｾﾝｻｰ 後退
      LD      M419  ; 初期SOL励磁
      AND     M203  ; IDｾﾝｻｰ前後 後退端
      ORB
      ANI     M505  ; IDｾﾝｻｰ 前進
      ORB
      AND     X0  ; 運転準備
      AND     M17  ; 運転モード切替
      OUT     M506  ; IDｾﾝｻｰ 後退
1113  LD      M505  ; IDｾﾝｻｰ 前進
      ANI     Y263  ; IDｾﾝｻｰ前後 後退 SOL
      OUT     Y262  ; IDｾﾝｻｰ前後 前進 SOL
1116  LD      M506  ; IDｾﾝｻｰ 後退
      ANI     Y262  ; IDｾﾝｻｰ前後 前進 SOL
      OUT     Y263  ; IDｾﾝｻｰ前後 後退 SOL
1119  LD      T180  ; IDｾﾝｻｰ前後 前進端
      AND     T154  ; ﾅｯﾄﾗﾝﾅｰ部ｽﾄｯﾊﾟｰ ﾊﾟﾚｯﾄ有り
      AND     M252  ; ﾅｯﾄﾗﾝﾅｰ部ｽﾄｯﾊﾟｰ原位置
      AND     M208  ; ﾊﾟﾚｯﾄ位置決め 端
      ANI     L310  ; ID読み込み完了
      AND     X0  ; 運転準備
      OUT     M510  ; ID読込条件
1126  LD      M510  ; ID読込条件
      ANI     M512  ; ID読込完了
      OUT     M511  ; ID読込ｽﾀｰﾄ
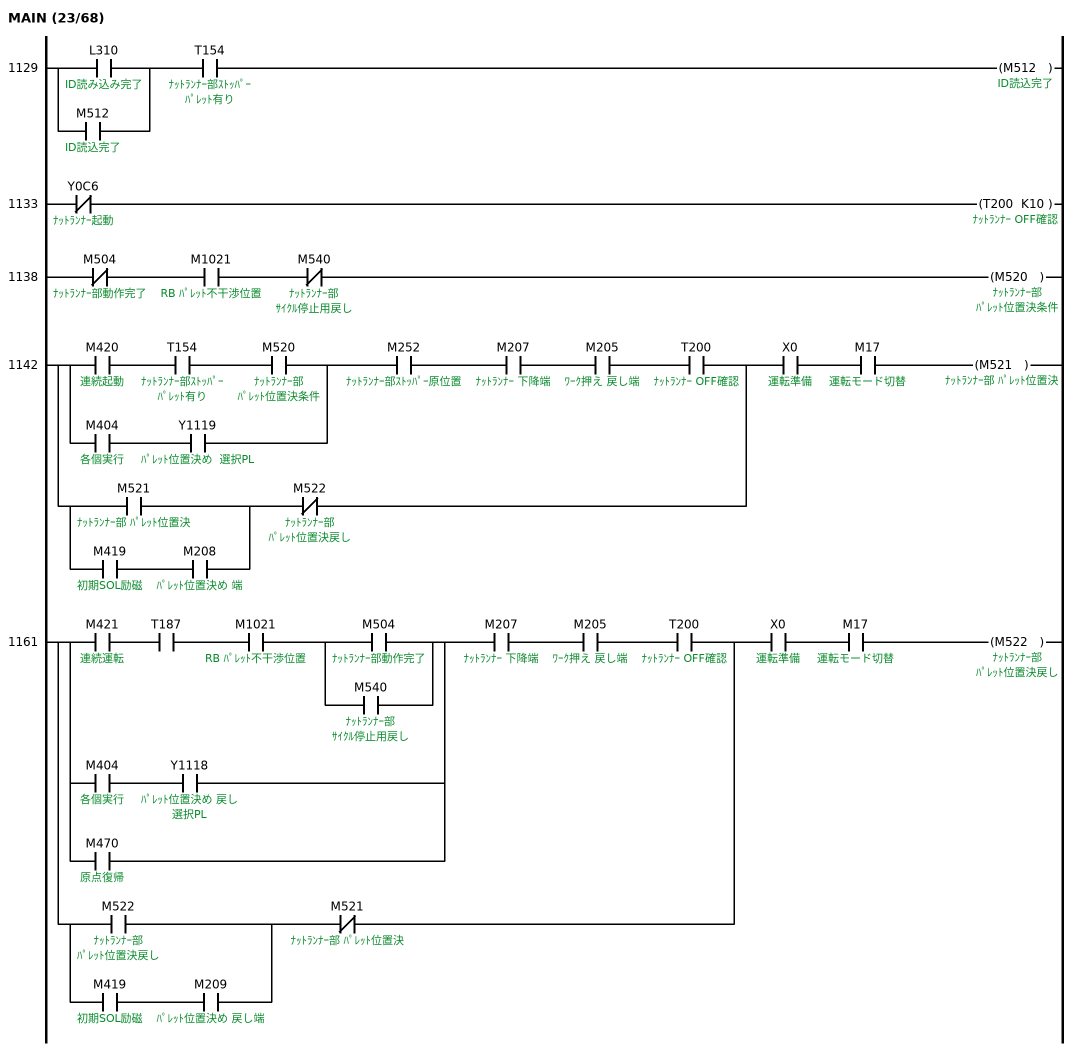
1129  LD      L310  ; ID読み込み完了
      OR      M512  ; ID読込完了
      AND     T154  ; ﾅｯﾄﾗﾝﾅｰ部ｽﾄｯﾊﾟｰ ﾊﾟﾚｯﾄ有り
      OUT     M512  ; ID読込完了
1133  LDI     Y0C6  ; ﾅｯﾄﾗﾝﾅｰ起動
      OUT     T200 K10  ; ﾅｯﾄﾗﾝﾅｰ OFF確認
1138  LDI     M504  ; ﾅｯﾄﾗﾝﾅｰ部動作完了
      AND     M1021  ; RB ﾊﾟﾚｯﾄ不干渉位置
      ANI     M540  ; ﾅｯﾄﾗﾝﾅｰ部 ｻｲｸﾙ停止用戻し
      OUT     M520  ; ﾅｯﾄﾗﾝﾅｰ部 ﾊﾟﾚｯﾄ位置決条件
1142  LD      M420  ; 連続起動
      AND     T154  ; ﾅｯﾄﾗﾝﾅｰ部ｽﾄｯﾊﾟｰ ﾊﾟﾚｯﾄ有り
      AND     M520  ; ﾅｯﾄﾗﾝﾅｰ部 ﾊﾟﾚｯﾄ位置決条件
      LD      M404  ; 各個実行
      AND     Y1119  ; ﾊﾟﾚｯﾄ位置決め  選択PL
      ORB
      AND     M252  ; ﾅｯﾄﾗﾝﾅｰ部ｽﾄｯﾊﾟｰ原位置
      AND     M207  ; ﾅｯﾄﾗﾝﾅｰ 下降端
      AND     M205  ; ﾜｰｸ押え 戻し端
      AND     T200  ; ﾅｯﾄﾗﾝﾅｰ OFF確認
      LD      M521  ; ﾅｯﾄﾗﾝﾅｰ部 ﾊﾟﾚｯﾄ位置決
      LD      M419  ; 初期SOL励磁
      AND     M208  ; ﾊﾟﾚｯﾄ位置決め 端
      ORB
      ANI     M522  ; ﾅｯﾄﾗﾝﾅｰ部 ﾊﾟﾚｯﾄ位置決戻し
      ORB
      AND     X0  ; 運転準備
      AND     M17  ; 運転モード切替
      OUT     M521  ; ﾅｯﾄﾗﾝﾅｰ部 ﾊﾟﾚｯﾄ位置決
1161  LD      M421  ; 連続運転
      AND     T187
      AND     M1021  ; RB ﾊﾟﾚｯﾄ不干渉位置
      LD      M504  ; ﾅｯﾄﾗﾝﾅｰ部動作完了
      OR      M540  ; ﾅｯﾄﾗﾝﾅｰ部 ｻｲｸﾙ停止用戻し
      ANB
      LD      M404  ; 各個実行
      AND     Y1118  ; ﾊﾟﾚｯﾄ位置決め 戻し 選択PL
      ORB
      OR      M470  ; 原点復帰
      AND     M207  ; ﾅｯﾄﾗﾝﾅｰ 下降端
      AND     M205  ; ﾜｰｸ押え 戻し端
      AND     T200  ; ﾅｯﾄﾗﾝﾅｰ OFF確認
      LD      M522  ; ﾅｯﾄﾗﾝﾅｰ部 ﾊﾟﾚｯﾄ位置決戻し
      LD      M419  ; 初期SOL励磁
      AND     M209  ; ﾊﾟﾚｯﾄ位置決め 戻し端
      ORB
      ANI     M521  ; ﾅｯﾄﾗﾝﾅｰ部 ﾊﾟﾚｯﾄ位置決
      ORB
      AND     X0  ; 運転準備
      AND     M17  ; 運転モード切替
      OUT     M522  ; ﾅｯﾄﾗﾝﾅｰ部 ﾊﾟﾚｯﾄ位置決戻し
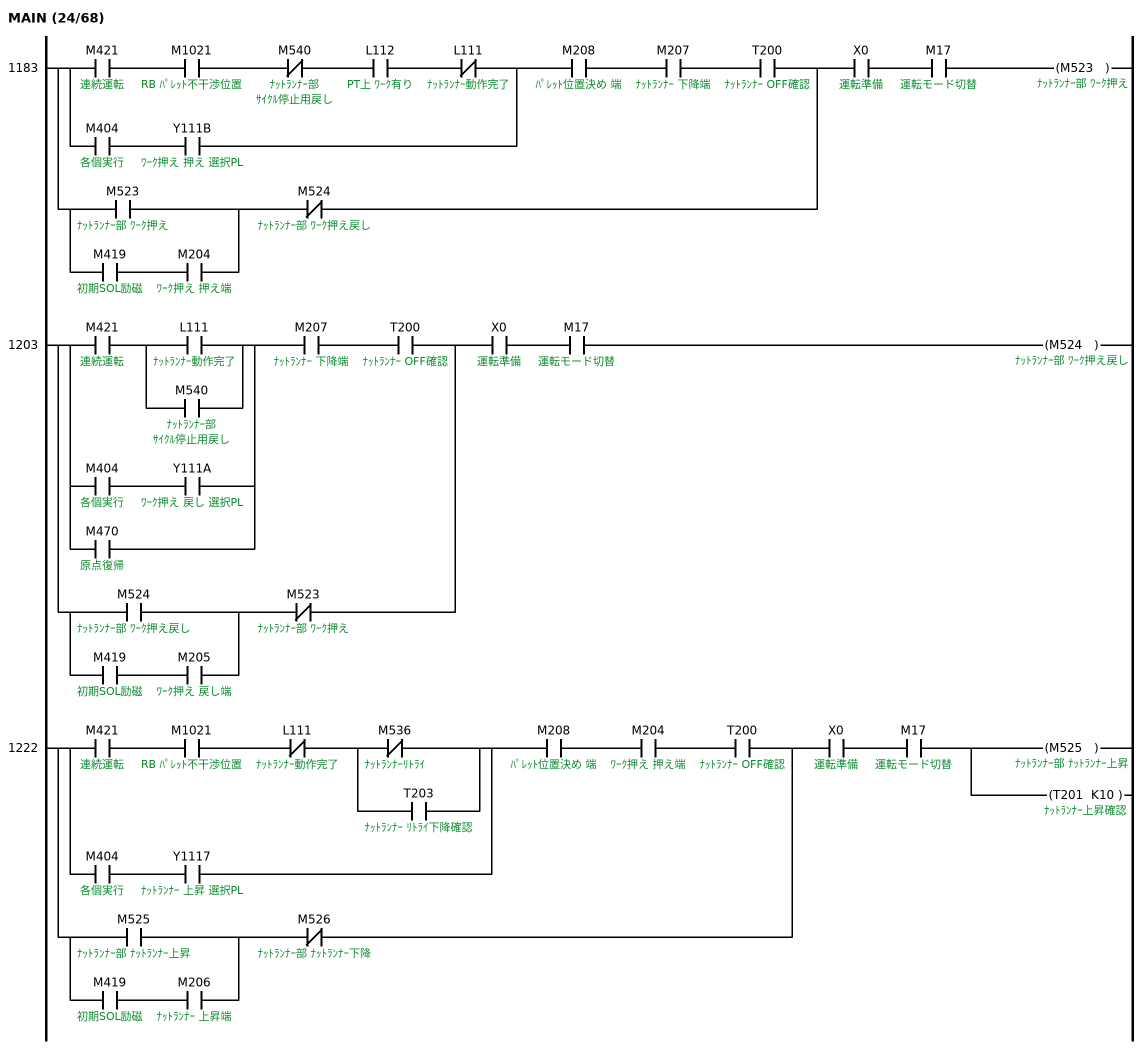
1183  LD      M421  ; 連続運転
      AND     M1021  ; RB ﾊﾟﾚｯﾄ不干渉位置
      ANI     M540  ; ﾅｯﾄﾗﾝﾅｰ部 ｻｲｸﾙ停止用戻し
      AND     L112  ; PT上 ﾜｰｸ有り
      ANI     L111  ; ﾅｯﾄﾗﾝﾅｰ動作完了
      LD      M404  ; 各個実行
      AND     Y111B  ; ﾜｰｸ押え 押え 選択PL
      ORB
      AND     M208  ; ﾊﾟﾚｯﾄ位置決め 端
      AND     M207  ; ﾅｯﾄﾗﾝﾅｰ 下降端
      AND     T200  ; ﾅｯﾄﾗﾝﾅｰ OFF確認
      LD      M523  ; ﾅｯﾄﾗﾝﾅｰ部 ﾜｰｸ押え
      LD      M419  ; 初期SOL励磁
      AND     M204  ; ﾜｰｸ押え 押え端
      ORB
      ANI     M524  ; ﾅｯﾄﾗﾝﾅｰ部 ﾜｰｸ押え戻し
      ORB
      AND     X0  ; 運転準備
      AND     M17  ; 運転モード切替
      OUT     M523  ; ﾅｯﾄﾗﾝﾅｰ部 ﾜｰｸ押え
1203  LD      M421  ; 連続運転
      LD      L111  ; ﾅｯﾄﾗﾝﾅｰ動作完了
      OR      M540  ; ﾅｯﾄﾗﾝﾅｰ部 ｻｲｸﾙ停止用戻し
      ANB
      LD      M404  ; 各個実行
      AND     Y111A  ; ﾜｰｸ押え 戻し 選択PL
      ORB
      OR      M470  ; 原点復帰
      AND     M207  ; ﾅｯﾄﾗﾝﾅｰ 下降端
      AND     T200  ; ﾅｯﾄﾗﾝﾅｰ OFF確認
      LD      M524  ; ﾅｯﾄﾗﾝﾅｰ部 ﾜｰｸ押え戻し
      LD      M419  ; 初期SOL励磁
      AND     M205  ; ﾜｰｸ押え 戻し端
      ORB
      ANI     M523  ; ﾅｯﾄﾗﾝﾅｰ部 ﾜｰｸ押え
      ORB
      AND     X0  ; 運転準備
      AND     M17  ; 運転モード切替
      OUT     M524  ; ﾅｯﾄﾗﾝﾅｰ部 ﾜｰｸ押え戻し
1222  LD      M421  ; 連続運転
      AND     M1021  ; RB ﾊﾟﾚｯﾄ不干渉位置
      ANI     L111  ; ﾅｯﾄﾗﾝﾅｰ動作完了
      LDI     M536  ; ﾅｯﾄﾗﾝﾅｰﾘﾄﾗｲ
      OR      T203  ; ﾅｯﾄﾗﾝﾅｰ ﾘﾄﾗｲ下降確認
      ANB
      LD      M404  ; 各個実行
      AND     Y1117  ; ﾅｯﾄﾗﾝﾅｰ 上昇 選択PL
      ORB
      AND     M208  ; ﾊﾟﾚｯﾄ位置決め 端
      AND     M204  ; ﾜｰｸ押え 押え端
      AND     T200  ; ﾅｯﾄﾗﾝﾅｰ OFF確認
      LD      M525  ; ﾅｯﾄﾗﾝﾅｰ部 ﾅｯﾄﾗﾝﾅｰ上昇
      LD      M419  ; 初期SOL励磁
      AND     M206  ; ﾅｯﾄﾗﾝﾅｰ 上昇端
      ORB
      ANI     M526  ; ﾅｯﾄﾗﾝﾅｰ部 ﾅｯﾄﾗﾝﾅｰ下降
      ORB
      AND     X0  ; 運転準備
      AND     M17  ; 運転モード切替
      OUT     M525  ; ﾅｯﾄﾗﾝﾅｰ部 ﾅｯﾄﾗﾝﾅｰ上昇
      OUT     T201 K10  ; ﾅｯﾄﾗﾝﾅｰ上昇確認
